TPL.FC_SetException(i_xExceptionActive	:= xUpdateStructsException, 
					iq_stException		:= stUpdateStructsException, 
					iq_stExceptionList	:= iq_stExceptionList, 
					iq_stLogDataList	:= iq_stLogDataList);
					
xInitSuccessful := xInitSuccessful AND NOT xUpdateStructsException;

etDiag := GD.ET_Diag.Ok;
(* End of system generated code, could be modified for your application *)
END_ACTION

END_PROGRAM

// LMC_PacDrive/Application/CrankModuleExample/Tools/FC_IsDriveVirtual
FUNCTION FC_IsDriveVirtual : BOOL
VAR_INPUT
	i_ifDrive	: SystemConfigurationItf.IF_Drive;
END_VAR

VAR_OUTPUT
	q_etDiag	: GD.ET_Diag := GD.ET_Diag.Ok;
	q_etDiagExt	: ET_DiagExt := ET_DiagExt.Ok;
	q_sMsg		: STRING[80];
END_VAR

VAR
	xSuccess						: BOOL;
	ifSercosDeviceIdentification	: SystemConfigurationItf.IF_SercosDeviceIdentification; 
END_VAR

IF i_ifDrive = 0 THEN
	q_etDiag	:= GD.ET_Diag.InputParameterInvalid;
	q_etDiagExt	:= ET_DiagExt.DriveInvalid;
	q_sMsg		:= 'FC_IsDriveVirtual: i_ifDrive not set';		
ELSE
	xSuccess := __QUERYINTERFACE(i_ifDrive, ifSercosDeviceIdentification);
	IF NOT xSuccess OR ifSercosDeviceIdentification = 0 THEN
		q_etDiag	:= GD.ET_Diag.InputParameterInvalid;
		q_etDiagExt	:= ET_DiagExt.DriveInvalid;
		q_sMsg		:= Standard.CONCAT(i_ifDrive.Name, ' - IF_SercosDeviceIdentification not implemented');						
	ELSE
		IF ifSercosDeviceIdentification.WorkingState = 0 THEN	// Drive is virtual
			FC_IsDriveVirtual := TRUE;
		ELSE
			FC_IsDriveVirtual := FALSE;
		END_IF
	END_IF
END_IF

END_FUNCTION

// LMC_PacDrive/Application/CrankModuleExample/Tools/FC_SetDeadTimeCompensation
FUNCTION FC_SetDeadTimeCompensation : BOOL
VAR_INPUT
	i_stSubModuleInterfaceMain		: AXM.ST_Main;
END_VAR
VAR
(* Init related variables *)	
	stLogicalAddressMaster			: SystemConfigurationItf.ST_LogicalAddress;
	lrShaftRefDelay					: LREAL;
	lrPositionDelay					: LREAL; 
	diResult						: DINT;	

END_VAR

IF i_stSubModuleInterfaceMain.i_ifMaster <> 0 AND i_stSubModuleInterfaceMain.i_ifDrive <> 0 THEN	
	stLogicalAddressMaster := i_stSubModuleInterfaceMain.i_ifMaster.stLogicalAddress;
	IF (stLogicalAddressMaster.udiType = SYSTEMINTERFACE.P_ENC_TYPE.udiType) OR			(* Physical encoder *)
		(stLogicalAddressMaster.udiType = SYSTEMINTERFACE.INC_IN_TYPE.udiType) OR		(* Incremental	encoder *)
		(stLogicalAddressMaster.udiType = SYSTEMINTERFACE.V_ENC_TYPE.udiType) THEN		(* Virtual master encoder *)
		
		stLogicalAddressMaster := i_stSubModuleInterfaceMain.i_ifDrive.stLogicalAddress;
		stLogicalAddressMaster.udiParameterId := 16#00A2;
		diResult := SYSTEMINTERFACE.FC_GetParameter(i_stLogAdr	:= stLogicalAddressMaster,
													i_dwBuffer	:= ADR(lrShaftRefDelay),
													i_diSize	:= SIZEOF(lrShaftRefDelay));
		IF diResult = 0 THEN
			i_stSubModuleInterfaceMain.iq_lencEncoder.Delay := -lrShaftRefDelay;
		END_IF
	ELSIF (stLogicalAddressMaster.udiType = SYSTEMINTERFACE.INC_IN3_TYPE.udiType) THEN  (* IncIn via TM5 TM5SE1IC20005 *)
		stLogicalAddressMaster := i_stSubModuleInterfaceMain.i_ifDrive.stLogicalAddress;
		stLogicalAddressMaster.udiParameterId := 16#00A2;
		diResult := SYSTEMINTERFACE.FC_GetParameter(i_stLogAdr	:= stLogicalAddressMaster,
													i_dwBuffer	:= ADR(lrShaftRefDelay),
													i_diSize	:= SIZEOF(lrShaftRefDelay));
		IF diResult = 0 THEN
			i_stSubModuleInterfaceMain.iq_lencEncoder.Delay := -lrShaftRefDelay;
			stLogicalAddressMaster := i_stSubModuleInterfaceMain.i_ifMaster.stLogicalAddress;
			stLogicalAddressMaster.udiParameterId := 16#008E; 					(* Parameter PositionDelay of TM5SE1IC20005 *)
			diResult := SYSTEMINTERFACE.FC_GetParameter(i_stLogAdr	:= stLogicalAddressMaster,
														i_dwBuffer	:= ADR(lrPositionDelay),
														i_diSize	:= SIZEOF(lrPositionDelay));		
			IF diResult = 0 THEN
				i_stSubModuleInterfaceMain.iq_lencEncoder.Delay := -(lrShaftRefDelay + (-lrPositionDelay)) ;
			END_IF
		END_IF
	END_IF
END_IF

IF diResult = 0 THEN
	FC_SetDeadTimeCompensation := TRUE;
END_IF

END_FUNCTION

// LMC_PacDrive/Application/CrankModuleExample/EquipmentModules/SR_BravoModule
PROGRAM SR_BravoModule

VAR CONSTANT
(* Standard related constants *)
	c_udiNumberOfGroups				: UDINT := 3;			(* Maximum number of groups *)
	c_udiNumberOfGroupMembers		: UDINT := 10;			(* Maximum number of members per group *)

	c_udiNumberOfCmdTables			: UDINT := 8;			(* Must be the exact number of used CMDTables! *)
	c_udiNumberOfCmdSteps			: UDINT := 16;			(* Make sure that the number of commands/ Steps  that each table
																   contains does not exceed the c_diNumberOfCMDSteps variable.*)

(* Definition group of modules *)
	c_udiBravoGroup1				: UDINT := 2001;		(* Name of module group  1 *)
	c_udiBravoGroup2				: UDINT := 2002;		(* Name of module group  2 *)

(* System generated code, could be modified for your application *)
	c_udiNumberOfSubModules			: UDINT := 2;			(* Number of axis modules *)
	c_udiSlave1						: UDINT := 1;
	c_udiSlave2						: UDINT := 2;
(* End of system generated code, could be modified for your application *)
END_VAR

VAR (* User specific variables *)
	stSlave1Interface				: AXM.ST_ModuleInterface;
	fbSlave1Module					: AXM.FB_AxisModule;
	
	stSlave2Interface				: AXM.ST_ModuleInterface;
	fbSlave2Module					: FB_AxisModuleExtItf;
	
	fbAxisModuleController			: AXM.FB_AxisModuleController;
END_VAR

VAR_INPUT
(* Master of BravoModule *)
	i_ifMaster						: SystemConfigurationItf.IF_Master;
END_VAR

VAR_IN_OUT
(* TPL.ST_StandardModuleInterface *)	
	iq_stStandardModuleItf			: TPL.ST_StandardModuleInterface;
	
(* TPL.ST_StandardMotionInterface *)		
	iq_stStandardMotionItf			: TPL.ST_StandardMotionInterface;
	
(* ExceptionHandling and Logging *)	
	iq_stExceptionList				: TPL.ST_ExceptionList;
	iq_stLogDataList				: TPL.ST_LogDataList;
END_VAR

VAR
	xInitSuccessful : BOOL := TRUE;
		
(* Standard related variables *)
	astSubModuleInterface			: ARRAY[1..c_udiNumberOfSubModules] OF TPL.ST_StandardModuleInterface;		(* Interface to modules *)
	aaudiSubModuleGroups			: ARRAY[1..c_udiNumberOfGroups,1..c_udiNumberOfGroupMembers] OF UDINT;
	adwSubModuleAddInterfaces		: ARRAY[1..c_udiNumberOfSubModules] OF DWORD;

(* Modules related variables *)
	fbModuleController				: TPL.FB_ModuleController;
	etDiagModuleController			: GD.ET_Diag;
	etDiagExtModuleController		: TPL.ET_DiagExt;
	sMsgModuleController			: STRING[80];
	xWaitForStartStep				: BOOL;
	
	astListOfCmdTables				: ARRAY [1..c_udiNumberOfCmdTables] OF TPL.ST_CmdTable;
	udiTableIndex					: UDINT;
	udiStepIndex					: UDINT;
	diStep							: DINT;

	astPrepareTable					: ARRAY [1..c_udiNumberOfCmdSteps] OF TPL.ST_Cmd;		(* Relating  Cmd table *)
	astAutoTable					: ARRAY [1..c_udiNumberOfCmdSteps] OF TPL.ST_Cmd;		(* Relating  Cmd table *)
	astManualTable					: ARRAY [1..c_udiNumberOfCmdSteps] OF TPL.ST_Cmd;		(* Relating  Cmd table *)
	astHoldTable					: ARRAY [1..c_udiNumberOfCmdSteps] OF TPL.ST_Cmd;		(* Relating  Cmd table *)
	astStartTable					: ARRAY [1..c_udiNumberOfCmdSteps] OF TPL.ST_Cmd;		(* Relating  Cmd table *)
	astStopTable					: ARRAY [1..c_udiNumberOfCmdSteps] OF TPL.ST_Cmd;		(* Relating  Cmd table *)
	astBrakeReleaseTable			: ARRAY [1..c_udiNumberOfCmdSteps] OF TPL.ST_Cmd;		(* Relating  Cmd table *)
	astAbortTable					: ARRAY [1..c_udiNumberOfCmdSteps] OF TPL.ST_Cmd;		(* Relating  Cmd table *)

(* ExceptionHandling related variables *)
	fbExceptionHandler				: TPL.FB_ExceptionHandler;

	aetReactionTranslationMode		: ARRAY[1..c_udiNumberOfSubModules] OF TPL.ET_ReactionTranslationMode;
	aastReactionTranslationTable	: ARRAY[1..c_udiNumberOfSubModules,1..TPL.Gc_udiMaxNumberOfReactions] OF TPL.ST_Reaction;
	astReactionTranslationJobs		: ARRAY[1..c_udiNumberOfSubModules] OF TPL.ST_ReactionTranslationJobs;
	
(* Exception declaration *)
	stUserException1				: TPL.ST_Exception;
	stUserException2				: TPL.ST_Exception;
	xModuleUserException1			: BOOL;
	xModuleUserException2			: BOOL;
	
	stUpdateStructsException		: TPL.ST_Exception;
	xUpdateStructsException			: BOOL;
	
	stInitReactionsException		: TPL.ST_Exception;
	xInitReactionsException			: BOOL;
	
	stInitSubModulesException		: TPL.ST_Exception;
	xInitSubModulesException		: BOOL;
	
	stIsDriveVirtualException		: TPL.ST_Exception;
	xIsDriveVirtualException		: BOOL;

(* Logging related variables *)
	fbLogger						: TPL.FB_Logger;

(* OnlineChange related variables *)
	fbDetectOnlineChange			: TPL.FB_DetectOnlineChange;
	xDetectOnlineChangeActive		: BOOL; 
	xDetectOnlineChangeReady		: BOOL; 
	etDetectOnlineChangeDiag		: GD.ET_Diag;
	etDetectOnlineChangeDiagExt		: TPL.ET_DiagExt; 
	sDetectOnlineChangeMsg			: STRING[80];
	
(* Init related variables *)	
	stLogicalAddressMaster			: SystemConfigurationItf.ST_LogicalAddress;
	lrShaftRefDelay					: LREAL;
	diResult						: DINT;	
	
	xDriveIsVirtual					: BOOL;	
	
(* POU-Feedback related variables *)	
	etDiag			: GD.ET_Diag;
	etDiagExt		: ET_DiagExt;
	etDiagExtTPL	: TPL.ET_DiagExt;
	etDiagExtAXM	: AXM.ET_DiagExt;
	sMsgBuffer		: STRING[80];
END_VAR

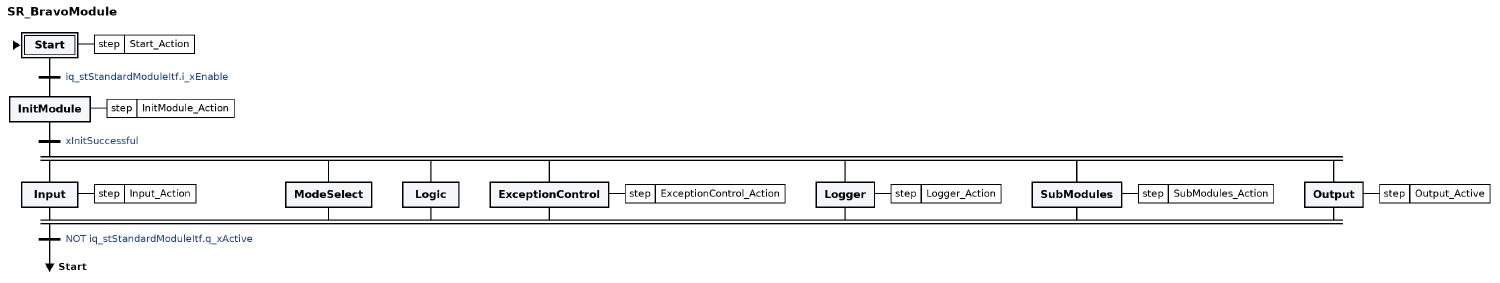
INITIAL_STEP Start:
    Start_Action(N);  // step action
END_STEP
TRANSITION FROM Start TO InitModule
    := iq_stStandardModuleItf.i_xEnable;
END_TRANSITION
STEP InitModule:
    InitModule_Action(N);  // step action
END_STEP
TRANSITION FROM InitModule TO (Input, ModeSelect, Logic, ExceptionControl, Logger, SubModules, Output)
    := xInitSuccessful;
END_TRANSITION
STEP Input:
    Input_Action(N);  // step action
END_STEP
STEP ModeSelect:
END_STEP
STEP Logic:
END_STEP
STEP ExceptionControl:
    ExceptionControl_Action(N);  // step action
END_STEP
STEP Logger:
    Logger_Action(N);  // step action
END_STEP
STEP SubModules:
    SubModules_Action(N);  // step action
END_STEP
STEP Output:
    Output_Active(N);  // step action
END_STEP
TRANSITION FROM (Input, ModeSelect, Logic, ExceptionControl, Logger, SubModules, Output) TO Start
    := NOT iq_stStandardModuleItf.q_xActive;
END_TRANSITION

ACTION ExceptionControl_Action:
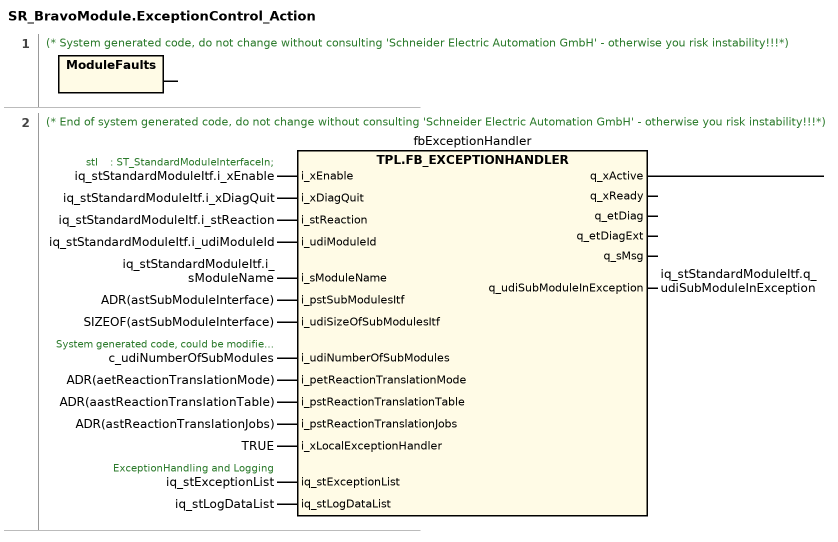
// NETWORK 1
// (* System generated code, do not change without consulting 'Schneider Electric Automation GmbH' - otherwise you risk instability!!!*)
ModuleFaults();

// NETWORK 2
// (* End of system generated code, do not change without consulting 'Schneider Electric Automation GmbH' - otherwise you risk instability!!!*)
//   fbExceptionHandler: ExceptionHandling related variables
//   iq_stStandardModuleItf.i_xEnable: stI : ST_StandardModuleInterfaceIn;
//   c_udiNumberOfSubModules: System generated code, could be modified for your application
//   iq_stExceptionList: ExceptionHandling and Logging
fbExceptionHandler(
    i_xEnable := iq_stStandardModuleItf.i_xEnable,
    i_xDiagQuit := iq_stStandardModuleItf.i_xDiagQuit,
    i_stReaction := iq_stStandardModuleItf.i_stReaction,
    i_udiModuleId := iq_stStandardModuleItf.i_udiModuleId,
    i_sModuleName := iq_stStandardModuleItf.i_sModuleName,
    i_pstSubModulesItf := ADR(astSubModuleInterface),
    i_udiSizeOfSubModulesItf := SIZEOF(astSubModuleInterface),
    i_udiNumberOfSubModules := c_udiNumberOfSubModules,
    i_petReactionTranslationMode := ADR(aetReactionTranslationMode),
    i_pstReactionTranslationTable := ADR(aastReactionTranslationTable),
    i_pstReactionTranslationJobs := ADR(astReactionTranslationJobs),
    i_xLocalExceptionHandler := TRUE,
    iq_stExceptionList := iq_stExceptionList,
    iq_stLogDataList := iq_stLogDataList,
    q_udiSubModuleInException => iq_stStandardModuleItf.q_udiSubModuleInException); // TPL.FB_EXCEPTIONHANDLER
END_ACTION

ACTION Init_CmdTables:
(* System generated code, could be modified for your application *)

(*********************************************************************************************************************)
(*** Prepare  ***)

TPL.FC_FirstStep(udiStepIndex, diStep);
astPrepareTable[udiStepIndex].sTitle					:= 'DriveEnable On AllSubModules';
astPrepareTable[udiStepIndex].udiModuleName				:= TPL.Gc_udiAllSubModules;
astPrepareTable[udiStepIndex].diStep					:= diStep;
astPrepareTable[udiStepIndex].diCMD						:= AXM.ET_Cmd.DriveEnableOn;
astPrepareTable[udiStepIndex].timTimeOut				:= T#0MS;
astPrepareTable[udiStepIndex].xEndCMD					:= FALSE;

TPL.FC_NextStep(udiStepIndex, diStep);
astPrepareTable[udiStepIndex].sTitle					:= 'Homing Mode AllSubModules';
astPrepareTable[udiStepIndex].udiModuleName				:= TPL.Gc_udiAllSubModules;
astPrepareTable[udiStepIndex].diStep					:= diStep;
astPrepareTable[udiStepIndex].diCMD						:= AXM.ET_Cmd.Homing;
astPrepareTable[udiStepIndex].timTimeOut				:= T#0MS;
astPrepareTable[udiStepIndex].xEndCMD					:= FALSE;

TPL.FC_NextStep(udiStepIndex, diStep);
astPrepareTable[udiStepIndex].sTitle					:= 'Homing Start AllSubModules';
astPrepareTable[udiStepIndex].udiModuleName				:= TPL.Gc_udiAllSubModules;
astPrepareTable[udiStepIndex].diStep					:= diStep;
astPrepareTable[udiStepIndex].diCMD						:= AXM.ET_Cmd.Start;
astPrepareTable[udiStepIndex].timTimeOut				:= T#0MS;
astPrepareTable[udiStepIndex].xEndCMD					:= FALSE;

TPL.FC_LastStep(udiStepIndex, diStep);
astPrepareTable[udiStepIndex].sTitle					:= 'End';
astPrepareTable[udiStepIndex].udiModuleName				:= 0;
astPrepareTable[udiStepIndex].diStep					:= diStep;
astPrepareTable[udiStepIndex].diCMD						:= 0;
astPrepareTable[udiStepIndex].timTimeOut				:= T#0MS;
astPrepareTable[udiStepIndex].xEndCMD					:= TRUE;

TPL.FC_FirstCmdTable(iq_udiTableIndex:= udiTableIndex);
astListofCMDTables[udiTableIndex].sTitle				:= 'Prepare';
astListofCMDTables[udiTableIndex].diCMD					:= ET_Cmd.Prepare;
astListofCMDTables[udiTableIndex].udiNumberOfCmdSteps	:= udiStepIndex;

(*********************************************************************************************************************)
(*** Auto  ***)

TPL.FC_FirstStep(udiStepIndex, diStep);
astAutoTable[udiStepIndex].sTitle						:= 'DriveEnable On AllSubModules';
astAutoTable[udiStepIndex].udiModuleName				:= TPL.Gc_udiAllSubModules;
astAutoTable[udiStepIndex].diStep						:= diStep;
astAutoTable[udiStepIndex].diCMD						:= AXM.ET_Cmd.DriveEnableOn;
astAutoTable[udiStepIndex].timTimeOut					:= T#0MS;
astAutoTable[udiStepIndex].xEndCMD						:= FALSE;

TPL.FC_NextStep(udiStepIndex, diStep);
astAutoTable[udiStepIndex].sTitle						:= 'Cam WS Mode AllSubModules';
astAutoTable[udiStepIndex].udiModuleName				:= TPL.Gc_udiAllSubModules;
astAutoTable[udiStepIndex].diStep						:= diStep;
astAutoTable[udiStepIndex].diCMD						:= AXM.ET_Cmd.CamWs;
astAutoTable[udiStepIndex].timTimeOut					:= T#0MS;
astAutoTable[udiStepIndex].xEndCMD						:= FALSE;

TPL.FC_NextStep(udiStepIndex, diStep);
astAutoTable[udiStepIndex].sTitle						:= 'Start AllSubModules';
astAutoTable[udiStepIndex].udiModuleName				:= TPL.Gc_udiAllSubModules;
astAutoTable[udiStepIndex].diStep						:= diStep;
astAutoTable[udiStepIndex].diCMD						:= AXM.ET_Cmd.Start;
astAutoTable[udiStepIndex].timTimeOut					:= T#0MS;
astAutoTable[udiStepIndex].xEndCMD						:= FALSE;

TPL.FC_NextStep(udiStepIndex, diStep);
astAutoTable[udiStepIndex].sTitle						:= 'WarmStart AllSubModules';
astAutoTable[udiStepIndex].udiModuleName				:= TPL.Gc_udiAllSubModules;
astAutoTable[udiStepIndex].diStep						:= diStep;
astAutoTable[udiStepIndex].diCMD						:= AXM.ET_Cmd.WsStart;
astAutoTable[udiStepIndex].timTimeOut					:= T#0MS;
astAutoTable[udiStepIndex].xEndCMD						:= FALSE;

TPL.FC_LastStep(udiStepIndex, diStep);
astAutoTable[udiStepIndex].sTitle						:= 'End';
astAutoTable[udiStepIndex].udiModuleName				:= 0;
astAutoTable[udiStepIndex].diStep						:= diStep;
astAutoTable[udiStepIndex].diCMD						:= 0;
astAutoTable[udiStepIndex].timTimeOut					:= T#0MS;
astAutoTable[udiStepIndex].xEndCMD						:= TRUE;

TPL.FC_NextCmdTable(iq_udiTableIndex:= udiTableIndex);
astListofCMDTables[udiTableIndex].sTitle				:= 'Auto';
astListofCMDTables[udiTableIndex].diCMD					:= ET_Cmd.Auto;
astListofCMDTables[udiTableIndex].udiNumberOfCmdSteps	:= udiStepIndex;

(*********************************************************************************************************************)
(*** Manual  ***)

TPL.FC_FirstStep(udiStepIndex, diStep);
astManualTable[udiStepIndex].sTitle						:= 'DriveEnable On AllSubModules';
astManualTable[udiStepIndex].udiModuleName				:= TPL.Gc_udiAllSubModules;
astManualTable[udiStepIndex].diStep						:= diStep;
astManualTable[udiStepIndex].diCMD						:= AXM.ET_Cmd.DriveEnableOn;
astManualTable[udiStepIndex].timTimeOut					:= T#0MS;
astManualTable[udiStepIndex].xEndCMD					:= FALSE;

TPL.FC_NextStep(udiStepIndex, diStep);
astManualTable[udiStepIndex].sTitle						:= 'Manual Mode AllSubModules';
astManualTable[udiStepIndex].udiModuleName				:= TPL.Gc_udiAllSubModules;
astManualTable[udiStepIndex].diStep						:= diStep;
astManualTable[udiStepIndex].diCMD						:= AXM.ET_Cmd.Manual;
astManualTable[udiStepIndex].timTimeOut					:= T#0MS;
astManualTable[udiStepIndex].xEndCMD					:= FALSE;

TPL.FC_LastStep(udiStepIndex, diStep);
astManualTable[udiStepIndex].sTitle						:= 'End';
astManualTable[udiStepIndex].udiModuleName				:= 0;
astManualTable[udiStepIndex].diStep						:= diStep;
astManualTable[udiStepIndex].diCMD						:= 0;
astManualTable[udiStepIndex].timTimeOut					:= T#0MS;
astManualTable[udiStepIndex].xEndCMD					:= TRUE;

TPL.FC_NextCmdTable(iq_udiTableIndex:= udiTableIndex);
astListofCMDTables[udiTableIndex].sTitle				:= 'Manual';
astListofCMDTables[udiTableIndex].diCMD					:= ET_Cmd.Manual;
astListofCMDTables[udiTableIndex].udiNumberOfCmdSteps	:= udiStepIndex;

(*********************************************************************************************************************)
(*** Stop ***)

TPL.FC_FirstStep(udiStepIndex, diStep);
astStopTable[udiStepIndex].sTitle						:= 'Stop AllSubModules';
astStopTable[udiStepIndex].udiModuleName				:= TPL.Gc_udiAllSubModules;
astStopTable[udiStepIndex].diStep						:= diStep;
astStopTable[udiStepIndex].diCMD						:= AXM.ET_Cmd.Stop;
astStopTable[udiStepIndex].timTimeOut					:= T#0MS;
astStopTable[udiStepIndex].xEndCMD						:= FALSE;

TPL.FC_LastStep(udiStepIndex, diStep);
astStopTable[udiStepIndex].sTitle						:= 'End';
astStopTable[udiStepIndex].udiModuleName				:= 0;
astStopTable[udiStepIndex].diStep						:= diStep;
astStopTable[udiStepIndex].diCMD						:= 0;
astStopTable[udiStepIndex].timTimeOut					:= T#0MS;
astStopTable[udiStepIndex].xEndCMD						:= TRUE;

TPL.FC_NextCmdTable(iq_udiTableIndex:= udiTableIndex);
astListofCMDTables[udiTableIndex].sTitle				:= 'Stop';
astListofCMDTables[udiTableIndex].diCMD					:= ET_Cmd.Stop;
astListofCMDTables[udiTableIndex].udiNumberOfCmdSteps	:= udiStepIndex;

(*********************************************************************************************************************)
(*** Start ***)

TPL.FC_FirstStep(udiStepIndex, diStep);
astStartTable[udiStepIndex].sTitle						:= 'Start AllSubModules';
astStartTable[udiStepIndex].udiModuleName				:= TPL.Gc_udiAllSubModules;
astStartTable[udiStepIndex].diStep						:= diStep;
astStartTable[udiStepIndex].diCMD						:= AXM.ET_Cmd.Start;
astStartTable[udiStepIndex].timTimeOut					:= T#0MS;
astStartTable[udiStepIndex].xEndCMD						:= FALSE;

TPL.FC_LastStep(udiStepIndex, diStep);
astStartTable[udiStepIndex].sTitle						:= 'End';
astStartTable[udiStepIndex].udiModuleName				:= 0;
astStartTable[udiStepIndex].diStep						:= diStep;
astStartTable[udiStepIndex].diCMD						:= 0;
astStartTable[udiStepIndex].timTimeOut					:= T#0MS;
astStartTable[udiStepIndex].xEndCMD						:= TRUE;

TPL.FC_NextCmdTable(iq_udiTableIndex:= udiTableIndex);
astListofCMDTables[udiTableIndex].sTitle				:= 'Start';
astListofCMDTables[udiTableIndex].diCMD					:= ET_Cmd.Start;
astListofCMDTables[udiTableIndex].udiNumberOfCmdSteps	:= udiStepIndex;

(*********************************************************************************************************************)
(*** Abort ***)

TPL.FC_FirstStep(udiStepIndex, diStep);
astAbortTable[udiStepIndex].sTitle						:= 'Stop AllSubModules';
astAbortTable[udiStepIndex].udiModuleName				:= TPL.Gc_udiAllSubModules;
astAbortTable[udiStepIndex].diStep						:= diStep;
astAbortTable[udiStepIndex].diCMD						:= AXM.ET_Cmd.Stop;
astAbortTable[udiStepIndex].timTimeOut					:= T#0MS;
astAbortTable[udiStepIndex].xEndCMD						:= FALSE;

TPL.FC_LastStep(udiStepIndex, diStep);
astAbortTable[udiStepIndex].sTitle						:= 	'End';
astAbortTable[udiStepIndex].udiModuleName				:= 	0;
astAbortTable[udiStepIndex].diStep						:= 	diStep;
astAbortTable[udiStepIndex].diCMD						:= 	0;
astAbortTable[udiStepIndex].timTimeOut					:=	T#0MS;
astAbortTable[udiStepIndex].xEndCMD						:= TRUE;

TPL.FC_NextCmdTable(iq_udiTableIndex:= udiTableIndex);
astListofCMDTables[udiTableIndex].sTitle				:= 'Abort';
astListofCMDTables[udiTableIndex].diCMD					:= ET_Cmd.Abort;
astListofCMDTables[udiTableIndex].udiNumberOfCmdSteps	:= udiStepIndex;

(*********************************************************************************************************************)
(*** Hold ***)

TPL.FC_FirstStep(udiStepIndex, diStep);
astHoldTable[udiStepIndex].sTitle						:= 'Hold AllSubModules';
astHoldTable[udiStepIndex].udiModuleName				:= TPL.Gc_udiAllSubModules;
astHoldTable[udiStepIndex].diStep						:= diStep;
astHoldTable[udiStepIndex].diCMD						:= AXM.ET_Cmd.Hold;
astHoldTable[udiStepIndex].timTimeOut					:= T#0MS;
astHoldTable[udiStepIndex].xEndCMD						:= FALSE;

TPL.FC_LastStep(udiStepIndex, diStep);
astHoldTable[udiStepIndex].sTitle						:= 'End';
astHoldTable[udiStepIndex].udiModuleName				:= 0;
astHoldTable[udiStepIndex].diStep						:= diStep;
astHoldTable[udiStepIndex].diCMD						:= 0;
astHoldTable[udiStepIndex].timTimeOut					:= T#0MS;
astHoldTable[udiStepIndex].xEndCMD						:= TRUE;

TPL.FC_NextCmdTable(iq_udiTableIndex:= udiTableIndex);
astListofCMDTables[udiTableIndex].sTitle				:= 'Hold';
astListofCMDTables[udiTableIndex].diCMD					:= ET_Cmd.Hold;
astListofCMDTables[udiTableIndex].udiNumberOfCmdSteps	:= udiStepIndex;

(*********************************************************************************************************************)
(*** Brake Release ***)

TPL.FC_FirstStep(udiStepIndex, diStep);
astBrakeReleaseTable[udiStepIndex].sTitle				:= 'AxisEnable Off AllSubModules';
astBrakeReleaseTable[udiStepIndex].udiModuleName		:= TPL.Gc_udiAllSubModules;
astBrakeReleaseTable[udiStepIndex].diStep				:= diStep;
astBrakeReleaseTable[udiStepIndex].diCMD				:= AXM.ET_Cmd.DriveEnableOff;
astBrakeReleaseTable[udiStepIndex].timTimeOut			:= T#0MS;
astBrakeReleaseTable[udiStepIndex].xEndCMD				:= FALSE;

TPL.FC_NextStep(udiStepIndex, diStep);
astBrakeReleaseTable[udiStepIndex].sTitle				:= 'BrakeRelease Mode AllSubModules';
astBrakeReleaseTable[udiStepIndex].udiModuleName		:= TPL.Gc_udiAllSubModules;
astBrakeReleaseTable[udiStepIndex].diStep				:= diStep;
astBrakeReleaseTable[udiStepIndex].diCMD				:= AXM.ET_Cmd.BrakeRelease;
astBrakeReleaseTable[udiStepIndex].timTimeOut			:= T#0MS;
astBrakeReleaseTable[udiStepIndex].xEndCMD				:= FALSE;

TPL.FC_NextStep(udiStepIndex, diStep);
astBrakeReleaseTable[udiStepIndex].sTitle				:= 'Start AllSubModules';
astBrakeReleaseTable[udiStepIndex].udiModuleName		:= TPL.Gc_udiAllSubModules;
astBrakeReleaseTable[udiStepIndex].diStep				:= diStep;
astBrakeReleaseTable[udiStepIndex].diCMD				:= AXM.ET_Cmd.Start;
astBrakeReleaseTable[udiStepIndex].timTimeOut			:= T#0MS;
astBrakeReleaseTable[udiStepIndex].xEndCMD				:= FALSE;

TPL.FC_LastStep(udiStepIndex, diStep);
astBrakeReleaseTable[udiStepIndex].sTitle				:= 'End';
astBrakeReleaseTable[udiStepIndex].udiModuleName		:= 0;
astBrakeReleaseTable[udiStepIndex].diStep				:= diStep;
astBrakeReleaseTable[udiStepIndex].diCMD				:= 0;
astBrakeReleaseTable[udiStepIndex].timTimeOut			:= T#0MS;
astBrakeReleaseTable[udiStepIndex].xEndCMD				:= TRUE;

TPL.FC_NextCmdTable(iq_udiTableIndex:= udiTableIndex);
astListofCMDTables[udiTableIndex].sTitle				:= 'Brake Release';
astListofCMDTables[udiTableIndex].diCMD					:= ET_Cmd.BrakeRelease;
astListofCMDTables[udiTableIndex].udiNumberOfCmdSteps	:= udiStepIndex;

(* End of system generated code, could be modified for your application *)
END_ACTION

ACTION Init_Exceptions:
(* System generated code, could be modified for your application *)
stUpdateStructsException.etDiag												:= GD.ET_Diag.UnexpectedProgramBehavior;
stUpdateStructsException.udiDiagExt											:= ET_DiagExt.UpdateStructsException;
stUpdateStructsException.sDiagExt											:= FC_EtDiagExtToString(i_etDiagExt := stUpdateStructsException.udiDiagExt);
stUpdateStructsException.sMsg												:= '';	(* Replaced on usage *)
stUpdateStructsException.udiModuleId										:= iq_stStandardModuleItf.i_udiModuleId;
stUpdateStructsException.sModuleName										:= iq_stStandardModuleItf.i_sModuleName;
stUpdateStructsException.stReaction.axReaction[TPL.ET_Reaction.AsyncStop]	:= TRUE;
stUpdateStructsException.etSource											:= TPL.ET_ExceptionSource.NodeModule;
stUpdateStructsException.timDelayTime										:= T#0MS;
stUpdateStructsException.wHmiAttributes										:= 0;
stUpdateStructsException.xAutoQuit											:= FALSE;

stInitReactionsException.etDiag												:= GD.ET_Diag.UnexpectedProgramBehavior;
stInitReactionsException.udiDiagExt											:= ET_DiagExt.InitReactionsException;
stInitReactionsException.sDiagExt											:= FC_EtDiagExtToString(i_etDiagExt := stInitReactionsException.udiDiagExt);
stInitReactionsException.sMsg												:= '';	(* Replaced on usage *)
stInitReactionsException.udiModuleId										:= iq_stStandardModuleItf.i_udiModuleId;
stInitReactionsException.sModuleName										:= iq_stStandardModuleItf.i_sModuleName;
stInitReactionsException.stReaction.axReaction[TPL.ET_Reaction.AsyncStop]	:= TRUE;
stInitReactionsException.etSource											:= TPL.ET_ExceptionSource.NodeModule;
stInitReactionsException.timDelayTime										:= T#0MS;
stInitReactionsException.wHmiAttributes										:= 0;
stInitReactionsException.xAutoQuit											:= FALSE;

stInitSubModulesException.etDiag											:= GD.ET_Diag.UnexpectedProgramBehavior;
stInitSubModulesException.udiDiagExt										:= ET_DiagExt.InitSubModulesException;
stInitSubModulesException.sDiagExt											:= FC_EtDiagExtToString(i_etDiagExt := stInitSubModulesException.udiDiagExt);
stInitSubModulesException.sMsg												:= '';	(* Replaced on usage *)
stInitSubModulesException.udiModuleId										:= iq_stStandardModuleItf.i_udiModuleId;
stInitSubModulesException.sModuleName										:= iq_stStandardModuleItf.i_sModuleName;
stInitSubModulesException.stReaction.axReaction[TPL.ET_Reaction.AsyncStop]	:= TRUE;
stInitSubModulesException.etSource											:= TPL.ET_ExceptionSource.NodeModule;
stInitSubModulesException.timDelayTime										:= T#0MS;
stInitSubModulesException.wHmiAttributes									:= 0;
stInitSubModulesException.xAutoQuit											:= FALSE;


(*------------------------------------------------------------------------------------------*)
(* Init User Exceptions *)

	// TPL.ET_Reaction.AsyncStop
	// TPL.ET_Reaction.SyncStopEL
	// TPL.ET_Reaction.SyncStopEH
	// TPL.ET_Reaction.StopEndOfCycle
	// TPL.ET_Reaction.MainsContactorOff
	
(*------------------------------------------------------------------------------------------*)
stUserException1.etDiag													:= GD.ET_Diag.ExecutionAborted;
stUserException1.udiDiagExt												:= ET_DiagExtUser.Exception1FromEquipmentModule;
stUserException1.sDiagExt												:= FC_EtDiagExtUserToString(i_etDiagExt := stUserException1.udiDiagExt);
stUserException1.sMsg													:= 'User Exception 1';
stUserException1.udiModuleId											:= iq_stStandardModuleItf.i_udiModuleId;
stUserException1.sModuleName											:= iq_stStandardModuleItf.i_sModuleName;
stUserException1.stReaction.axReaction[TPL.Gc_udiUserReactionOffset+2]	:= TRUE;
stUserException1.etSource												:= TPL.ET_ExceptionSource.User;
stUserException1.timDelayTime											:= T#0MS;
stUserException1.wHmiAttributes											:= 0;
stUserException1.xAutoQuit												:= FALSE;

stUserException2.etDiag													:= GD.ET_Diag.ExecutionAborted;
stUserException2.udiDiagExt												:= ET_DiagExtUser.Exception2FromEquipmentModule;
stUserException2.sDiagExt												:= FC_EtDiagExtUserToString(i_etDiagExt := stUserException2.udiDiagExt);
stUserException2.sMsg													:= 'User Exception 2';
stUserException2.udiModuleId											:= iq_stStandardModuleItf.i_udiModuleId;
stUserException2.sModuleName											:= iq_stStandardModuleItf.i_sModuleName;
stUserException2.stReaction.axReaction[TPL.Gc_udiUserReactionOffset+2]	:= TRUE;
stUserException2.etSource												:= TPL.ET_ExceptionSource.User;
stUserException2.timDelayTime											:= T#0MS;
stUserException2.wHmiAttributes											:= 0;
stUserException2.xAutoQuit												:= FALSE;

(* End of system generated code, could be modified for your application *)
END_ACTION

ACTION Init_Reactions:
(* System generated code, only to be changed by experienced programmers *)
IF c_udiNumberOfSubModules < 1 THEN
	RETURN;
END_IF

(* Change of default reactions only on demand *)
(* Compare SR MainMachine Action Init_Reactions *)

xInitReactionsException := FALSE;

(*****************************************************************************************************************************************************)
(* Init ReactionTranslationMode *)

TPL.FC_InitReactionTranslationMode(	i_udiNumberOfSubModules			:= c_udiNumberOfSubModules,
									i_petReactionTranslationMode	:= ADR(aetReactionTranslationMode),
									q_etDiag						=> etDiag,
									q_etDiagExt						=> etDiagExtTPL);
							
IF etDiag <> GD.ET_Diag.Ok AND NOT xInitReactionsException THEN
	xInitReactionsException := TRUE;
	
	stInitReactionsException.sMsg := PDL.FC_MultiConcat(i_sString1 := 'InitReactionTranslationMode - ', 
														i_sString2 := GD.FC_EtDiagToString(i_etDiag := etDiag), 
														i_sString3 := ' - ', 
														i_sString4 := TPL.FC_EtDiagExtToString(i_etDiagExt := etDiagExtTPL));
END_IF	

(*****************************************************************************************************************************************************)
(* Init ReactionTranslationTable *)	

TPL.FC_InitReactionTranslationTable(i_udiNumberOfSubModules			:= c_udiNumberOfSubModules,
									i_pstReactionTranslationTable	:= ADR(aastReactionTranslationTable),
									q_etDiag						=> etDiag,
									q_etDiagExt						=> etDiagExtTPL);
									
IF etDiag <> GD.ET_Diag.Ok AND NOT xInitReactionsException THEN
	xInitReactionsException := TRUE;
	
	stInitReactionsException.sMsg := PDL.FC_MultiConcat(i_sString1 := 'InitReactionTranslationTable - ', 
														i_sString2 := GD.FC_EtDiagToString(i_etDiag := etDiag), 
														i_sString3 := ' - ', 
														i_sString4 := TPL.FC_EtDiagExtToString(i_etDiagExt := etDiagExtTPL));
END_IF		

(*****************************************************************************************************************************************************)
(* Init ReactionTranslationJobs *)	
								
TPL.FC_InitReactionTranslationJobs( i_udiNumberOfSubModules			:= c_udiNumberOfSubModules,
									i_pstReactionTranslationJobs	:= ADR(astReactionTranslationJobs),
									q_etDiag						=> etDiag,
									q_etDiagExt						=> etDiagExtTPL);
						
IF etDiag <> GD.ET_Diag.Ok AND NOT xInitReactionsException THEN
	xInitReactionsException := TRUE;
	
	stInitReactionsException.sMsg := PDL.FC_MultiConcat(i_sString1 := 'InitReactionTranslationJobs - ', 
														i_sString2 := GD.FC_EtDiagToString(i_etDiag := etDiag), 
														i_sString3 := ' - ', 
														i_sString4 := TPL.FC_EtDiagExtToString(i_etDiagExt := etDiagExtTPL));
END_IF		

(*****************************************************************************************************************************************************)
(* Set exception if any exception occurred *)

TPL.FC_SetException(i_xExceptionActive	:= xInitReactionsException, 
					iq_stException		:= stInitReactionsException, 
					iq_stExceptionList	:= iq_stExceptionList, 
					iq_stLogDataList	:= iq_stLogDataList);
					
xInitSuccessful := xInitSuccessful AND NOT xInitReactionsException;

etDiag := GD.ET_Diag.Ok;
(* End of system generated code, only to be changed by experienced programmers *)
END_ACTION

ACTION Init_Slave1:
(* System generated code, could be modified for your application *)

(* Standard interface *)
astSubModuleInterface[c_udiSlave1].i_sModuleName		:= CONCAT(STR1 := iq_stStandardModuleItf.i_sModuleName, STR2 := ': Slave1');

astSubModuleInterface[c_udiSlave1].i_xLogEnable			:= 	TRUE;
astSubModuleInterface[c_udiSlave1].i_wLogDataFilter		:= 	UDINT_TO_WORD(TPL.ET_LogDataFilter.ModuleDefault);

(* AxisModule specific interface *)
stSlave1Interface.stMain.i_ifMaster			:= i_ifMaster; 		(* Master *)
stSlave1Interface.stMain.i_ifDrive			:= DRV_Slave1;
stSlave1Interface.stMain.iq_lencEncoder		:= LE_Slave1;


xDriveIsVirtual := FC_IsDriveVirtual(	i_ifDrive	:= stSlave1Interface.stMain.i_ifDrive,
										q_etDiag	=> etDiag,
										q_etDiagExt	=> etDiagExt, //etDiagExtTPL,
										q_sMsg		=> sMsgBuffer);

IF etDiag <> GD.ET_Diag.Ok AND NOT xIsDriveVirtualException THEN										
	stIsDriveVirtualException.sMsg := sMsgBuffer;
	xIsDriveVirtualException := TRUE;
END_IF

TPL.FC_SetException(i_xExceptionActive	:= xIsDriveVirtualException, 
					iq_stException		:= stIsDriveVirtualException, 
					iq_stExceptionList	:= iq_stExceptionList, 
					iq_stLogDataList	:= iq_stLogDataList);
					
xInitSuccessful := xInitSuccessful AND NOT xIsDriveVirtualException;
etDiag := GD.ET_Diag.Ok;
	

(*Set DeadTime compensation parameters depending on used type of Master*)
FC_SetDeadTimeCompensation(i_stSubModuleInterfaceMain := stSlave1Interface.stMain);
  (*Please note, FC_DeadTimeCompensation does not recognize the master type, transferred via C2C or encoder network! 
	stXXXXInterface.stMain.iq_lencEncoder.Delay must be adjusted in order to reach shaft synchronism, it depends on:
	- Transmission delay via the choosen network, depending on topology and timing 
	- Type of the master e.g. physical encoder or an axis
	- SERCOS cycle times in master and slave controllers
	
	C2C sample (similar for encoder network):
	//Access C2C_EncIn.DataDelay only if C2C_Master.SyncGroupState=5 or C2C_Slave.SyncGroupState = 5 and C2C_EncIn.DataValid = TRUE!

		//Master is a physical encoder (PMEnc/Inc):
			stXXXXInterface.stMain.iq_lencEncoder.Delay := C2C_EncIn.DataDelay - DRV_SlaveAxis.ShaftRefDelay;

		//Master is an axis (real/ virtual):
			stXXXXInterface.stMain.iq_lencEncoder.Delay := C2C_EncIn.DataDelay + one SERCOS cycle of C2C controller with connected master axis;*)


stSlave1Interface.stMain.i_lrMotionActiveVelLimit						:= 15.0;	(* Limit for max. velocity of astAxisModuleInterface to switch output AxisMove in Units/s *)
stSlave1Interface.stMain.i_etMotionActiveVelType						:= AXM.ET_MotionActiveVelType.Velocity;

stSlave1Interface.stMain.i_timMasterStop								:= T#1S;
stSlave1Interface.stMain.i_xHwLimitPos									:= FALSE;
stSlave1Interface.stMain.i_xHwLimitNeg									:= FALSE;

stSlave1Interface.stMain.stReducedVelocity.i_xEnableReducedVelocity		:= FALSE;
stSlave1Interface.stMain.stReducedVelocity.i_xOnlyLimitCheck			:= FALSE;
stSlave1Interface.stMain.stReducedVelocity.i_lrMaxReducedVelocity		:= 50.0;

stSlave1Interface.stMain.i_xStart										:= FALSE;

(***************************************************************************************************************************************************************************************************)

(*** Homing ***)

IF xDriveIsVirtual THEN
	stSlave1Interface.stHome.i_etMode := PDL.ET_HomeMode.SetPosAxisAndLogEncoderPosition;			(* Homing Mode  in case of virtual axis *)
ELSE
	stSlave1Interface.stHome.i_etMode := PDL.ET_HomeMode.PosDirectionPosEdgeTp;						(* Homing Mode in case of real axis *)
END_IF
	

stSlave1Interface.stHome.i_xEnableInitAbsReadPos := FALSE;		(* TRUE : Restores the AxisPosition depending on the stHome.etMode
																		  If stHome.i_etMode is equal to PDL.ET_HomeMode.RestorePosFromAxisEncoder or 
																		  to PDL.ET_HomeMode.WriteAxisEncoder, the encoder of the axis is read,
																		  or else the position will be restored from the retain area *)
																		  
stSlave1Interface.stHome.stSetpos.iq_pstRestorePosRetain := ADR(Grp_stRestorePositionAxis2);

stSlave1Interface.stHome.i_xResetHomeOk := FALSE;

(* Possible modes for homing mode Sensor:
	PDL.ET_HomeMode.PosDirectionPosEdgeSensor
	PDL.ET_HomeMode.NegDirectionPosEdgeSensor
	PDL.ET_HomeMode.NegDirectionNegEdgeSensor
	PDL.ET_HomeMode.PosDirectionNegEdgeSensor
*)
stSlave1Interface.stHome.stSensor.i_lrHomePosition			:= 0.0;			(* Position at the end of homing in units *)
stSlave1Interface.stHome.stSensor.i_lrVel					:= 10.0;		(* Homing ceiling velocity in units/s *)
stSlave1Interface.stHome.stSensor.i_lrAcc					:= 1000.0;		(* Homing acceleration in units/s^2 *)
stSlave1Interface.stHome.stSensor.i_lrDec					:= 1000.0;		(* Homing deceleration in units/s^2 *)
stSlave1Interface.stHome.stSensor.i_lrJerk					:= 10000.0;		(* Homing jerk in units/s^3 *)
stSlave1Interface.stHome.stSensor.i_lrOffset				:= 0.0;			(* Offset from home signal in units *)
stSlave1Interface.stHome.stSensor.i_lrMaxTravel				:= 720.0;		(* Max. travel for referencing by normal input *)
stSlave1Interface.stHome.stSensor.i_xRotativeSystem			:= FALSE;		(* Rotative system true or false for referencing by normal input *)
stSlave1Interface.stHome.stSensor.i_xSensor					:= FALSE;		(* Input for home signal. Can be a signal from a controller input. Has to be written cyclic. *)

(* Possible Modes for homing mode LimitSwitch:
	PDL.ET_HomeMode.PosDirectionPosEdgeHWLimitPos		normally open contact / Closing contact
	PDL.ET_HomeMode.NegDirectionPosEdgeHWLimitNeg		normally open contact / Closing contact
	PDL.ET_HomeMode.NegDirectionNegEdgeHWLimitNeg		normally closed contact / Opening contact  
	PDL.ET_HomeMode.PosDirectionNegEdgeHWLimitPos		normally closed contact / Opening contact 
*)
stSlave1Interface.stHome.stLimitSwitch.i_lrHomePosition		:= 0.0;			(* Position at the end of homing in units *)
stSlave1Interface.stHome.stLimitSwitch.i_lrVel				:= 10.0;		(* Homing ceiling velocity in units/s *)
stSlave1Interface.stHome.stLimitSwitch.i_lrLowVel			:= 5.0;			(* Homing low ceiling velocity in units/s *)
stSlave1Interface.stHome.stLimitSwitch.i_lrAcc				:= 1000.0;		(* Homing acceleration in units/s^2 *)
stSlave1Interface.stHome.stLimitSwitch.i_lrDec				:= 1000.0;		(* Homing deceleration in units/s^2 *)
stSlave1Interface.stHome.stLimitSwitch.i_lrJerk				:= 10000.0;		(* Homing jerk in units/s^3 *)
stSlave1Interface.stHome.stLimitSwitch.i_lrOffset			:= 0.0;			(* Offset from home signal in units *)
stSlave1Interface.stHome.stLimitSwitch.i_lrMaxTravel		:= 9999.0;		(* Max. travel for referencing normal input as a hardware limit *)

(* Possible modes for homing mode MoveOnPos:
	PDL.ET_HomeMode.MoveOnPosAbs 
*)
stSlave1Interface.stHome.stMoveOnPos.i_lrTarget				:= 0.0;			(* Position at the end of homing in units *)
stSlave1Interface.stHome.stMoveOnPos.i_lrVel				:= 10.0;		(* Homing ceiling velocity in units/s *)
stSlave1Interface.stHome.stMoveOnPos.i_lrAcc				:= 1000.0;		(* Homing acceleration in units/s^2 *)
stSlave1Interface.stHome.stMoveOnPos.i_lrDec				:= 1000.0;		(* Homing deceleration in units/s^2 *)
stSlave1Interface.stHome.stMoveOnPos.i_lrJerk				:= 10000.0;		(* Homing jerk in units/s^3 *)
stSlave1Interface.stHome.stMoveOnPos.i_lrPeriod				:= 0.0;			(* Period of the axis *)
stSlave1Interface.stHome.stMoveOnPos.i_xRotativeSystem		:= FALSE;		(* Rotative system true or false *)

(* Possible modes for homing mode SetPos:
	PDL.ET_HomeMode.SetPosAxisPosition 
	PDL.ET_HomeMode.SetPosLogEncoderPosition 
	PDL.ET_HomeMode.SetPosAxisAndLogEncoderPosition
	PDL.ET_HomeMode.RestorePosFromAxisEncoder 
	PDL.ET_HomeMode.RestorePosFromRetain 
*)
stSlave1Interface.stHome.stSetpos.i_lrHomePosition			:= 0.0;			(* Position at the end of homing in units *)
stSlave1Interface.stHome.stSetpos.i_lrEncoderPosition		:= 0.0;			(* Encoder position in units after homing *)
stSlave1Interface.stHome.stSetpos.i_lrAbsEncOffset			:= 100.0;		(* Distance to the jump of axis encoder in units  *)
stSlave1Interface.stHome.stSetpos.i_lrRestoreWindow			:= 180;			(* How far can the drive be away from is correct position *)
stSlave1Interface.stHome.stSetpos.i_lrUserPeriod			:= 360;			(* Period of the axis *)

(* Possible modes for homing mode Torque:
	PDL.ET_HomeMode.PosDirectionMaxTorque 
	PDL.ET_HomeMode.NegDirectionMaxTorque 
*)
stSlave1Interface.stHome.stTorque.i_lrHomePosition			:= 0.0;			(* Position at the end of homing in units *)
stSlave1Interface.stHome.stTorque.i_lrVel					:= 10.0;		(* Homing ceiling velocity in units/s *)
stSlave1Interface.stHome.stTorque.i_lrAcc					:= 1000.0;		(* Homing acceleration in units/s^2 *)
stSlave1Interface.stHome.stTorque.i_lrDec					:= 1000.0;		(* Homing deceleration in units/s^2 *)
stSlave1Interface.stHome.stTorque.i_lrJerk					:= 10000.0;		(* Homing jerk in units/s^3 *)
stSlave1Interface.stHome.stTorque.i_lrOffset				:= 0.0;			(* Offset from home signal in units *)
stSlave1Interface.stHome.stTorque.i_lrMaxTravel				:= 9999.0;		(* Max. travel for referencing by torque *)
stSlave1Interface.stHome.stTorque.i_lrMaxTorque				:= 0.0;			(* Torque for stop in Nm / referencing by torque *)
stSlave1Interface.stHome.stTorque.i_diTorqueTime			:= 5;			(* Time in msec to hold torque *)

(* Possible modes for homing mode TouchProbe:
	PDL.ET_HomeMode.PosDirectionPosEdgeTp 
	PDL.ET_HomeMode.NegDirectionPosEdgeTp 
	PDL.ET_HomeMode.NegDirectionNegEdgeTp 
	PDL.ET_HomeMode.PosDirectionNegEdgeTp 
*)
stSlave1Interface.stHome.stTouchProbe.i_lrHomePosition		:= 0.0;			(* Position at the end of homing in units *)
stSlave1Interface.stHome.stTouchProbe.i_lrVel				:= 100.0;		(* Homing ceiling velocity in units/s *)
stSlave1Interface.stHome.stTouchProbe.i_lrAcc				:= 1000.0;		(* Homing acceleration in units/s^2 *)
stSlave1Interface.stHome.stTouchProbe.i_lrDec				:= 1000.0;		(* Homing deceleration in units/s^2 *)
stSlave1Interface.stHome.stTouchProbe.i_lrJerk				:= 10000.0;		(* Homing jerk in units/s^3 *)
stSlave1Interface.stHome.stTouchProbe.i_lrOffset			:= 30.0;		(* Offset from home signal in units *)
stSlave1Interface.stHome.stTouchProbe.i_lrMaxTravel			:= 720.0;		(* Max. travel for referencing by TP *)
stSlave1Interface.stHome.stTouchProbe.i_xRotativeSystem		:= TRUE;		(* Rotative system true or false for referencing by TP *)
stSlave1Interface.stHome.stTouchProbe.i_ifTouchProbe		:= TP_1;		(* Input for TP *)

(* Possible modes for homing mode WritePos:
	PDL.ET_HomeMode.WriteAxisEncoder 
*)
stSlave1Interface.stHome.stWritePos.i_lrHomePosition		:= 0.0;			(* Position at the end of homing in units *)
stSlave1Interface.stHome.stWritePos.i_lrUserPeriod			:= 0.0;			(* Calculates Drive.Position into period ( units ) *)
stSlave1Interface.stHome.stWritePos.i_lrAbsEncOffset		:= 100.0;		(* Distance to the jump of axis encoder in units *)

(***************************************************************************************************************************************************************************************************)
(*** Manual ***)

stSlave1Interface.stManual.i_lrVel								:= 50.0;			(* Velocity in units/s *)
stSlave1Interface.stManual.i_lrAcc								:= 100.0;			(* Acceleration in units/s^2 *)
stSlave1Interface.stManual.i_lrDec								:= 100.0;			(* Deceleration in units/s^2 *)
stSlave1Interface.stManual.i_lrJerk								:= 1000.0;			(* Jerk in units/s^3 *)
stSlave1Interface.stManual.i_lrMaxDistance						:= 120.0;			(* Max pathlengths for one step in units *)
stSlave1Interface.stManual.i_xEndless							:= FALSE;			(* TRUE: jogging endless; Position between the periode; FALSE: jogging in steps. Position can be out of periode *)
stSlave1Interface.stManual.i_lrPeriod							:= 360.0;			(* Period of the axis *)

(***************************************************************************************************************************************************************************************************)
(*** Cam ***)

stSlave1Interface.stMultiCam.i_etCSModeSlave					:= PDL.ET_MultiCamCsModeSlave.SetSlavePositionToFirstCamPosition;		(* ColdStartMode Slave *)
stSlave1Interface.stMultiCam.i_etCSModeMaster					:= PDL.ET_MultiCamCsModeMaster.SetMasterPositionToFirstCamPosition;		(* ColdStartMode Master *)
stSlave1Interface.stMultiCam.i_etWSMode							:= PDL.ET_MultiCamWsMode.StoredCamMoveAlwaysNoPositionCheck;			(* WarmStartMode *)
stSlave1Interface.stMultiCam.i_lrWSWindow						:= 5.0;											(* WarmStartWindow in Axis units *)
stSlave1Interface.stMultiCam.i_lrWSVel							:= 100.0;										(* Velocity for WarmStart and CSModeSlave = PDL.ET_MultiCamCsModeSlave.MoveSlaveToFirstCamPosition in Units/s *)
stSlave1Interface.stMultiCam.i_lrWSAcc							:= 1000.0;										(* Acceleration and deceleration for Warmstart and CSModeSlave = PDL.ET_MultiCamCsModeSlave.MoveSlaveToFirstCamPosition in Units/s^2 *)
stSlave1Interface.stMultiCam.i_lrWSJerk							:= 10000.0;										(* Jerk for Warmstart and CSModeSlave = PDL.ET_MultiCamCsModeSlave.MoveSlaveToFirstCamPosition in units/s^3 *)
stSlave1Interface.stMultiCam.i_diTXend							:= 2*SYSTEMINTERFACE.FC_LzsTaskGetInterval();	(* Time of XLowEnd and XHighEnd befor Xend or Xstart in msec*)
stSlave1Interface.stMultiCam.i_lrInstantXLimMax					:= 0.0;											(* Switch off position at 'InstantNewCam' *)

stSlave1Interface.stMultiCam.i_xEnableTabHandler				:= TRUE;										(* TRUE: TabHandler is enabled *)
stSlave1Interface.stMultiCam.i_udiTableSelectNr					:= AXM.ET_ParId.User;							(* Number of table which is used in the next cycle *)

stSlave1Interface.stMultiCam.i_xSetEncoderParameters			:= FALSE;										(* TRUE: The parameters MasterId, FeedConstand, GearIn and GearOut will be copyed into LEnc object *)
stSlave1Interface.stMultiCam.i_xSetEncoderPosition				:= FALSE;										(* TRUE: Manipulation of LEnc object on startup OpMode MultiCam *)
stSlave1Interface.stMultiCam.i_lrSetEncoderOffset				:= 0.0;											(* Master encoder offset *)
stSlave1Interface.stMultiCam.i_xCheckEncoderPeriod				:= TRUE;										(* TRUE: Check of encoder period = 0. If encoder period <> 0 -> Exception *)

stSlave1Interface.stMultiCam.iq_astMotionPar[AXM.ET_ParId.User].diNumberOfCamPoints		:= 4;	(* DataStruct for the next cycle *)
stSlave1Interface.stMultiCam.iq_astMotionPar[AXM.ET_ParId.User].lrYPeriod				:= 0.0;

stSlave1Interface.stMultiCam.iq_astMotionPar[AXM.ET_ParId.User].astCamPoint[0].lrX		:= 0.0;
stSlave1Interface.stMultiCam.iq_astMotionPar[AXM.ET_ParId.User].astCamPoint[0].lrY		:= 0.0;
stSlave1Interface.stMultiCam.iq_astMotionPar[AXM.ET_ParId.User].astCamPoint[0].lrM		:= 0.0;
stSlave1Interface.stMultiCam.iq_astMotionPar[AXM.ET_ParId.User].astCamPoint[0].etCamType	:= PDL.ET_CamType.Poly5Com;
stSlave1Interface.stMultiCam.iq_astMotionPar[AXM.ET_ParId.User].astCamPoint[1].lrX		:= 60.0;
stSlave1Interface.stMultiCam.iq_astMotionPar[AXM.ET_ParId.User].astCamPoint[1].lrY		:= 30.0;
stSlave1Interface.stMultiCam.iq_astMotionPar[AXM.ET_ParId.User].astCamPoint[1].lrM		:= 1.0;
stSlave1Interface.stMultiCam.iq_astMotionPar[AXM.ET_ParId.User].astCamPoint[1].etCamType	:= PDL.ET_CamType.Straight;
stSlave1Interface.stMultiCam.iq_astMotionPar[AXM.ET_ParId.User].astCamPoint[2].lrX		:= 240.0;
stSlave1Interface.stMultiCam.iq_astMotionPar[AXM.ET_ParId.User].astCamPoint[2].lrY		:= 210.0;
stSlave1Interface.stMultiCam.iq_astMotionPar[AXM.ET_ParId.User].astCamPoint[2].lrM		:= 1.0;
stSlave1Interface.stMultiCam.iq_astMotionPar[AXM.ET_ParId.User].astCamPoint[2].etCamType	:= PDL.ET_CamType.Poly5Com;
stSlave1Interface.stMultiCam.iq_astMotionPar[AXM.ET_ParId.User].astCamPoint[3].lrX		:= 360.0;
stSlave1Interface.stMultiCam.iq_astMotionPar[AXM.ET_ParId.User].astCamPoint[3].lrY		:= 0.0;
stSlave1Interface.stMultiCam.iq_astMotionPar[AXM.ET_ParId.User].astCamPoint[3].lrM		:= 0.0;
stSlave1Interface.stMultiCam.iq_astMotionPar[AXM.ET_ParId.User].astCamPoint[3].etCamType	:= PDL.ET_CamType.Poly5Com;

stSlave1Interface.stMultiCam.iq_astMotionPar[AXM.ET_ParId.Idle].diUserTableId	:= UDINT_TO_DINT(AXM.ET_ParId.Idle);
stSlave1Interface.stMultiCam.iq_astMotionPar[AXM.ET_ParId.Start].diUserTableId	:= UDINT_TO_DINT(AXM.ET_ParId.Start);
stSlave1Interface.stMultiCam.iq_astMotionPar[AXM.ET_ParId.Cont].diUserTableId	:= UDINT_TO_DINT(AXM.ET_ParId.Cont);
stSlave1Interface.stMultiCam.iq_astMotionPar[AXM.ET_ParId.Stop].diUserTableId	:= UDINT_TO_DINT(AXM.ET_ParId.Stop);
stSlave1Interface.stMultiCam.iq_astMotionPar[AXM.ET_ParId.User].diUserTableId	:= UDINT_TO_DINT(AXM.ET_ParId.User);

(***************************************************************************************************************************************************************************************************)
(*** Endless ***)

stSlave1Interface.stEndless.i_lrVel								:= 100.0;			(* Velocity in Units/s *)
stSlave1Interface.stEndless.i_lrAcc								:= 1000.0;			(* Acceleration in Units/s^2 *)
stSlave1Interface.stEndless.i_lrDec								:= 1000.0;			(* Deceleration in Units/s^2 *)
stSlave1Interface.stEndless.i_lrJerk							:= 10000.0;			(* Jerk in units/s^3 *)
stSlave1Interface.stEndless.i_lrPeriod							:= 360.0;			(* Period one cycle in units *)
stSlave1Interface.stEndless.i_lrStopPosition					:= 0.5;				(* Stop position in units *)


(***************************************************************************************************************************************************************************************************)
(*** Pos ***)

stSlave1Interface.stPos.i_etPosMode								:= SYSTEMINTERFACE.ET_PosMode.Relative;			(* SYSTEMINTERFACE.ET_PosMode.Endless, SYSTEMINTERFACE.ET_PosMode.Relative, SYSTEMINTERFACE.ET_PosMode.Absolute *)
stSlave1Interface.stPos.i_lrTarget								:= -360.0;										(* Target position or distance in Units *)
stSlave1Interface.stPos.i_lrVel									:= 100.0;										(* Ceiling velocity in Units/s *)
stSlave1Interface.stPos.i_lrAcc									:= 3600.0;										(* Acceleration in Units/s^2 *)
stSlave1Interface.stPos.i_lrDec									:= 3600.0;										(* Deceleration in Units/s^2 *)
stSlave1Interface.stPos.i_lrJerk								:= 36000.0;										(* Jerk in units/s^3 *)

(* End of system generated code, could be modified for your application *)
END_ACTION

ACTION Init_Slave2:
(* System generated code, could be modified for your application *)

(* Standard interface *)
astSubModuleInterface[c_udiSlave2].i_sModuleName	:= 	CONCAT(STR1 := iq_stStandardModuleItf.i_sModuleName, STR2 := ': Slave2');

astSubModuleInterface[c_udiSlave2].i_xLogEnable		:= 	TRUE;
astSubModuleInterface[c_udiSlave2].i_wLogDataFilter	:= 	UDINT_TO_WORD(TPL.ET_LogDataFilter.ModuleDefault);

(* AxisModule specific interface *)
stSlave2Interface.stMain.i_ifMaster		:= i_ifMaster; 		(* Master *)
stSlave2Interface.stMain.i_ifDrive		:= DRV_Slave2;
stSlave2Interface.stMain.iq_lencEncoder	:= LE_Slave2;


xDriveIsVirtual := FC_IsDriveVirtual(	i_ifDrive	:= stSlave2Interface.stMain.i_ifDrive,
										q_etDiag	=> etDiag,
										q_etDiagExt	=> etDiagExt,//etDiagExtTPL,
										q_sMsg		=> sMsgBuffer);

IF etDiag <> GD.ET_Diag.Ok AND NOT xIsDriveVirtualException THEN										
	stIsDriveVirtualException.sMsg := sMsgBuffer;
	xIsDriveVirtualException := TRUE;
END_IF

TPL.FC_SetException(i_xExceptionActive	:= xIsDriveVirtualException, 
					iq_stException		:= stIsDriveVirtualException, 
					iq_stExceptionList	:= iq_stExceptionList, 
					iq_stLogDataList	:= iq_stLogDataList);
					
xInitSuccessful := xInitSuccessful AND NOT xIsDriveVirtualException;
etDiag := GD.ET_Diag.Ok;
	

(*Set DeadTime compensation parameters depending on used type of Master*)
FC_SetDeadTimeCompensation(i_stSubModuleInterfaceMain := stSlave2Interface.stMain);
  (*Please note, FC_DeadTimeCompensation does not recognize the master type, transferred via C2C or encoder network! 
	stXXXXInterface.stMain.iq_lencEncoder.Delay must be adjusted in order to reach shaft synchronism, it depends on:
	- Transmission delay via the choosen network, depending on topology and timing 
	- Type of the master e.g. physical encoder or an axis
	- SERCOS cycle times in master and slave controllers
	
	C2C sample (similar for encoder network):
	//Access C2C_EncIn.DataDelay only if C2C_Master.SyncGroupState=5 or C2C_Slave.SyncGroupState = 5 and C2C_EncIn.DataValid = TRUE!

		//Master is a physical encoder (PMEnc/Inc):
			stXXXXInterface.stMain.iq_lencEncoder.Delay := C2C_EncIn.DataDelay - DRV_SlaveAxis.ShaftRefDelay;

		//Master is an axis (real/ virtual):
			stXXXXInterface.stMain.iq_lencEncoder.Delay := C2C_EncIn.DataDelay + one SERCOS cycle of C2C controller with connected master axis;*)


stSlave2Interface.stMain.i_lrMotionActiveVelLimit						:= 15.0;	(* Limit for max. velocity of astAxisModuleInterface to switch output AxisMove in Units/s *)
stSlave2Interface.stMain.i_etMotionActiveVelType						:= AXM.ET_MotionActiveVelType.Velocity;

stSlave2Interface.stMain.i_timMasterStop								:= T#1S;
stSlave2Interface.stMain.i_xHwLimitPos									:= FALSE;
stSlave2Interface.stMain.i_xHwLimitNeg									:= FALSE;

stSlave2Interface.stMain.stReducedVelocity.i_xEnableReducedVelocity		:= FALSE;
stSlave2Interface.stMain.stReducedVelocity.i_xOnlyLimitCheck			:= FALSE;
stSlave2Interface.stMain.stReducedVelocity.i_lrMaxReducedVelocity		:= 50.0;

stSlave2Interface.stMain.i_xStart										:= FALSE;

(***************************************************************************************************************************************************************************************************)

(*** Homing ***)

IF xDriveIsVirtual THEN
	stSlave2Interface.stHome.i_etMode := PDL.ET_HomeMode.SetPosAxisAndLogEncoderPosition;			(* Homing Mode  in case of virtual axis *)
ELSE
	stSlave2Interface.stHome.i_etMode := PDL.ET_HomeMode.PosDirectionPosEdgeTp;						(* Homing Mode in case of real axis *)
END_IF


stSlave2Interface.stHome.i_xEnableInitAbsReadPos := FALSE;		(* TRUE : Restores the AxisPosition depending on the stHome.etMode
																		  If stHome.i_etMode is equal to PDL.ET_HomeMode.RestorePosFromAxisEncoder or 
																		  to PDL.ET_HomeMode.WriteAxisEncoder, the encoder of the axis is read,
																		  or else the position will be restored from the retain area *)
																								 
stSlave2Interface.stHome.stSetpos.iq_pstRestorePosRetain := ADR(Grp_stRestorePositionAxis3);

stSlave2Interface.stHome.i_xResetHomeOk := FALSE;

(* Possible modes for homing mode Sensor:
	PDL.ET_HomeMode.PosDirectionPosEdgeSensor
	PDL.ET_HomeMode.NegDirectionPosEdgeSensor
	PDL.ET_HomeMode.NegDirectionNegEdgeSensor
	PDL.ET_HomeMode.PosDirectionNegEdgeSensor
*)
stSlave2Interface.stHome.stSensor.i_lrHomePosition			:= 0.0;			(* Position at the end of homing in units *)
stSlave2Interface.stHome.stSensor.i_lrVel					:= 10.0;		(* Homing ceiling velocity in units/s *)
stSlave2Interface.stHome.stSensor.i_lrAcc					:= 1000.0;		(* Homing acceleration in units/s^2 *)
stSlave2Interface.stHome.stSensor.i_lrDec					:= 1000.0;		(* Homing deceleration in units/s^2 *)
stSlave2Interface.stHome.stSensor.i_lrJerk					:= 10000.0;		(* Homing jerk in units/s^3 *)
stSlave2Interface.stHome.stSensor.i_lrOffset				:= 0.0;			(* Offset from home signal in units *)
stSlave2Interface.stHome.stSensor.i_lrMaxTravel				:= 720.0;		(* Max. travel for referencing by normal input *)
stSlave2Interface.stHome.stSensor.i_xRotativeSystem			:= FALSE;		(* Rotative system true or false for referencing by normal input *)
stSlave2Interface.stHome.stSensor.i_xSensor					:= FALSE;		(* Input for home signal. Can be a signal from a controller input. Has to be written cyclic. *)

(* Possible Modes for homing mode LimitSwitch:
	PDL.ET_HomeMode.PosDirectionPosEdgeHWLimitPos		normally open contact / Closing contact
	PDL.ET_HomeMode.NegDirectionPosEdgeHWLimitNeg		normally open contact / Closing contact
	PDL.ET_HomeMode.NegDirectionNegEdgeHWLimitNeg		normally closed contact / Opening contact  
	PDL.ET_HomeMode.PosDirectionNegEdgeHWLimitPos		normally closed contact / Opening contact 
*)
stSlave2Interface.stHome.stLimitSwitch.i_lrHomePosition		:= 0.0;			(* Position at the end of homing in units *)
stSlave2Interface.stHome.stLimitSwitch.i_lrVel				:= 10.0;		(* Homing ceiling velocity in units/s *)
stSlave2Interface.stHome.stLimitSwitch.i_lrLowVel			:= 5.0;			(* Homing low ceiling velocity in units/s *)
stSlave2Interface.stHome.stLimitSwitch.i_lrAcc				:= 1000.0;		(* Homing acceleration in units/s^2 *)
stSlave2Interface.stHome.stLimitSwitch.i_lrDec				:= 1000.0;		(* Homing deceleration in units/s^2 *)
stSlave2Interface.stHome.stLimitSwitch.i_lrJerk				:= 10000.0;		(* Homing jerk in units/s^3 *)	
stSlave2Interface.stHome.stLimitSwitch.i_lrOffset			:= 0.0;			(* Offset from home signal in units *)
stSlave2Interface.stHome.stLimitSwitch.i_lrMaxTravel		:= 9999.0;		(* Max. travel for referencing normal input as a hardware limit *)

(* Possible modes for homing mode MoveOnPos:
	PDL.ET_HomeMode.MoveOnPosAbs 
*)
stSlave2Interface.stHome.stMoveonPos.i_lrTarget				:= 0.0;			(* Position at the end of homing in units *)
stSlave2Interface.stHome.stMoveonPos.i_lrVel				:= 10.0;		(* Homing ceiling velocity in units/s *)
stSlave2Interface.stHome.stMoveonPos.i_lrAcc				:= 1000.0;		(* Homing acceleration in units/s^2 *)
stSlave2Interface.stHome.stMoveonPos.i_lrDec				:= 1000.0;		(* Homing deceleration in units/s^2 *)
stSlave2Interface.stHome.stMoveonPos.i_lrJerk				:= 10000.0;		(* Homing jerk in units/s^3 *)
stSlave2Interface.stHome.stMoveonPos.i_lrPeriod				:= 0.0;			(* Period of the axis *)
stSlave2Interface.stHome.stMoveonPos.i_xRotativeSystem		:= FALSE;		(* Rotative system true or false *)

(* Possible modes for homing mode SetPos:
	PDL.ET_HomeMode.SetPosAxisPosition 
	PDL.ET_HomeMode.SetPosLogEncoderPosition 
	PDL.ET_HomeMode.SetPosAxisAndLogEncoderPosition
	PDL.ET_HomeMode.RestorePosFromAxisEncoder 
	PDL.ET_HomeMode.RestorePosFromRetain 
*)
stSlave2Interface.stHome.stSetpos.i_lrHomePosition			:= 0.0;			(* Position at the end of homing in units *)
stSlave2Interface.stHome.stSetpos.i_lrEncoderPosition		:= 0.0;			(* Encoder position in units after homing *)
stSlave2Interface.stHome.stSetpos.i_lrAbsEncOffset			:= 100.0;		(* Distance to the jump of axis encoder in units  *)
stSlave2Interface.stHome.stSetpos.i_lrRestoreWindow			:= 180;			(* How far can the drive be away from is correct position *)
stSlave2Interface.stHome.stSetpos.i_lrUserPeriod			:= 360;			(* Period of the axis *)

(* Possible modes for homing mode Torque:
	PDL.ET_HomeMode.PosDirectionMaxTorque 
	PDL.ET_HomeMode.NegDirectionMaxTorque 
*)
stSlave2Interface.stHome.stTorque.i_lrHomePosition			:= 0.0;			(* Position at the end of homing in units *)
stSlave2Interface.stHome.stTorque.i_lrVel					:= 10.0;		(* Homing ceiling velocity in units/s *)
stSlave2Interface.stHome.stTorque.i_lrAcc					:= 1000.0;		(* Homing acceleration in units/s^2 *)
stSlave2Interface.stHome.stTorque.i_lrDec					:= 1000.0;		(* Homing deceleration in units/s^2 *)
stSlave2Interface.stHome.stTorque.i_lrJerk					:= 10000.0;		(* Homing jerk in units/s^3 *)
stSlave2Interface.stHome.stTorque.i_lrOffset				:= 0.0;			(* Offset from home signal in units *)
stSlave2Interface.stHome.stTorque.i_lrMaxTravel				:= 9999.0;		(* Max. travel for referencing by torque *)
stSlave2Interface.stHome.stTorque.i_lrMaxTorque				:= 0.0;			(* Torque for stop in Nm / referencing by torque *)
stSlave2Interface.stHome.stTorque.i_diTorqueTime			:= 5;			(* Time in msec to hold torque *)

(* Possible modes for homing mode TouchProbe:
	PDL.ET_HomeMode.PosDirectionPosEdgeTp 
	PDL.ET_HomeMode.NegDirectionPosEdgeTp 
	PDL.ET_HomeMode.NegDirectionNegEdgeTp 
	PDL.ET_HomeMode.PosDirectionNegEdgeTp 
*)
stSlave2Interface.stHome.stTouchProbe.i_lrHomePosition		:= 0.0;			(* Position at the end of homing in units *)
stSlave2Interface.stHome.stTouchProbe.i_lrVel				:= 100.0;		(* Homing ceiling velocity in units/s *)
stSlave2Interface.stHome.stTouchProbe.i_lrAcc				:= 1000.0;		(* Homing acceleration in units/s^2 *)
stSlave2Interface.stHome.stTouchProbe.i_lrDec				:= 1000.0;		(* Homing deceleration in units/s^2 *)
stSlave2Interface.stHome.stTouchProbe.i_lrJerk				:= 10000.0;		(* Homing jerk in units/s^3 *)
stSlave2Interface.stHome.stTouchProbe.i_lrOffset			:= 30.0;		(* Offset from home signal in units *)
stSlave2Interface.stHome.stTouchProbe.i_lrMaxTravel			:= 720.0;		(* Max. travel for referencing by TP *)
stSlave2Interface.stHome.stTouchProbe.i_xRotativeSystem		:= TRUE;		(* Rotative system true or false for referencing by TP *)
stSlave2Interface.stHome.stTouchProbe.i_ifTouchProbe		:= TP_2;		(* Input for TP *)

(* Possible modes for homing mode WritePos:
	PDL.ET_HomeMode.WriteAxisEncoder 
*)
stSlave2Interface.stHome.stWritePos.i_lrHomePosition		:= 0.0;			(* Position at the end of homing in units *)
stSlave2Interface.stHome.stWritePos.i_lrUserPeriod			:= 0.0;			(* Calculates Drive.position into period ( units ) *)
stSlave2Interface.stHome.stWritePos.i_lrAbsEncOffset		:= 100.0;		(* Distance to the jump of axis encoder in units *)

(***************************************************************************************************************************************************************************************************)
(*** Manual ***)

stSlave2Interface.stManual.i_lrVel								:= 50.0;			(* Velocity in units/s *)
stSlave2Interface.stManual.i_lrAcc								:= 100.0;			(* Acceleration in units/s^2 *)
stSlave2Interface.stManual.i_lrDec								:= 100.0;			(* Deceleration in units/s^2 *)
stSlave2Interface.stManual.i_lrJerk								:= 1000.0;			(* Jerk in units/s^3 *)
stSlave2Interface.stManual.i_lrMaxDistance						:= 120.0;			(* Max pathlengths for one step in units *)
stSlave2Interface.stManual.i_xEndless							:= FALSE;			(* TRUE: jogging endless; Position between the periode; FALSE: jogging in steps. Position can be out of periode *)
stSlave2Interface.stManual.i_lrPeriod							:= 360.0;			(* Period of the axis *)

(***************************************************************************************************************************************************************************************************)
(*** Cam ***)

stSlave2Interface.stMultiCam.i_etCSModeSlave					:= PDL.ET_MultiCamCsModeSlave.SetSlavePositionToFirstCamPosition;		(* ColdStartMode Slave *)
stSlave2Interface.stMultiCam.i_etCSModeMaster					:= PDL.ET_MultiCamCsModeMaster.SetMasterPositionToFirstCamPosition;		(* ColdStartMode Master *)
stSlave2Interface.stMultiCam.i_etWSMode							:= PDL.ET_MultiCamWsMode.StoredCamMoveAlwaysNoPositionCheck;			(* WarmStartMode *)
stSlave2Interface.stMultiCam.i_lrWSWindow						:= 5.0;											(* WarmStartWindow in Axis units *)
stSlave2Interface.stMultiCam.i_lrWSVel							:= 100.0;										(* Velocity for WarmStart and CSModeSlave = PDL.ET_MultiCamCsModeSlave.MoveSlaveToFirstCamPosition in Units/s *)
stSlave2Interface.stMultiCam.i_lrWSAcc							:= 1000.0;										(* Acceleration and deceleration for Warmstart and CSModeSlave = PDL.ET_MultiCamCsModeSlave.MoveSlaveToFirstCamPosition in Units/s^2 *)
stSlave2Interface.stMultiCam.i_lrWSJerk							:= 10000.0;										(* Jerk for Warmstart and CSModeSlave = PDL.ET_MultiCamCsModeSlave.MoveSlaveToFirstCamPosition in units/s^3 *)
stSlave2Interface.stMultiCam.i_diTXend							:= 2*SYSTEMINTERFACE.FC_LzsTaskGetInterval();	(* Time of XLowEnd and XHighEnd befor Xend or Xstart in msec*)
stSlave2Interface.stMultiCam.i_lrInstantXLimMax					:= 0.0;											(* Switch off position at 'InstantNewCam' *)

stSlave2Interface.stMultiCam.i_xEnableTabHandler				:= TRUE;										(* TRUE: TabHandler is enabled *)
stSlave2Interface.stMultiCam.i_udiTableSelectNr					:= AXM.ET_ParId.User;							(* Number of table which is used in the next cycle *)								

stSlave2Interface.stMultiCam.i_xSetEncoderParameters			:= FALSE;										(* TRUE: The parameters MasterId, FeedConstand, GearIn and GearOut will be copyed into LEnc object *)
stSlave2Interface.stMultiCam.i_xSetEncoderPosition				:= FALSE;										(* TRUE: Manipulation of LEnc object on startup OpMode MultiCam *)
stSlave2Interface.stMultiCam.i_lrSetEncoderOffset				:= 0.0;											(* Master encoder offset *)
stSlave2Interface.stMultiCam.i_xCheckEncoderPeriod				:= TRUE;										(* TRUE: Check of encoder period = 0. If encoder period <> 0 -> Exception *)

stSlave2Interface.stMultiCam.iq_astMotionPar[AXM.ET_ParId.User].diNumberOfCamPoints		:= 4;	(* DataStruct for the next cycle *)
stSlave2Interface.stMultiCam.iq_astMotionPar[AXM.ET_ParId.User].lrYPeriod				:= 0.0;

stSlave2Interface.stMultiCam.iq_astMotionPar[AXM.ET_ParId.User].astCamPoint[0].lrX		:= 0.0;
stSlave2Interface.stMultiCam.iq_astMotionPar[AXM.ET_ParId.User].astCamPoint[0].lrY		:= 0.0;
stSlave2Interface.stMultiCam.iq_astMotionPar[AXM.ET_ParId.User].astCamPoint[0].lrM		:= 0.0;
stSlave2Interface.stMultiCam.iq_astMotionPar[AXM.ET_ParId.User].astCamPoint[0].etCamType	:= PDL.ET_CamType.Poly5Com;
stSlave2Interface.stMultiCam.iq_astMotionPar[AXM.ET_ParId.User].astCamPoint[1].lrX		:= 60.0;
stSlave2Interface.stMultiCam.iq_astMotionPar[AXM.ET_ParId.User].astCamPoint[1].lrY		:= 30.0;
stSlave2Interface.stMultiCam.iq_astMotionPar[AXM.ET_ParId.User].astCamPoint[1].lrM		:= 1.0;
stSlave2Interface.stMultiCam.iq_astMotionPar[AXM.ET_ParId.User].astCamPoint[1].etCamType	:= PDL.ET_CamType.Straight;
stSlave2Interface.stMultiCam.iq_astMotionPar[AXM.ET_ParId.User].astCamPoint[2].lrX		:= 240.0;
stSlave2Interface.stMultiCam.iq_astMotionPar[AXM.ET_ParId.User].astCamPoint[2].lrY		:= 210.0;
stSlave2Interface.stMultiCam.iq_astMotionPar[AXM.ET_ParId.User].astCamPoint[2].lrM		:= 1.0;
stSlave2Interface.stMultiCam.iq_astMotionPar[AXM.ET_ParId.User].astCamPoint[2].etCamType	:= PDL.ET_CamType.Poly5Com;
stSlave2Interface.stMultiCam.iq_astMotionPar[AXM.ET_ParId.User].astCamPoint[3].lrX		:= 360.0;
stSlave2Interface.stMultiCam.iq_astMotionPar[AXM.ET_ParId.User].astCamPoint[3].lrY		:= 0.0;
stSlave2Interface.stMultiCam.iq_astMotionPar[AXM.ET_ParId.User].astCamPoint[3].lrM		:= 0.0;
stSlave2Interface.stMultiCam.iq_astMotionPar[AXM.ET_ParId.User].astCamPoint[3].etCamType	:= PDL.ET_CamType.Poly5Com;

stSlave2Interface.stMultiCam.iq_astMotionPar[AXM.ET_ParId.Idle].diUserTableId	:= UDINT_TO_DINT(AXM.ET_ParId.Idle);
stSlave2Interface.stMultiCam.iq_astMotionPar[AXM.ET_ParId.Start].diUserTableId	:= UDINT_TO_DINT(AXM.ET_ParId.Start);
stSlave2Interface.stMultiCam.iq_astMotionPar[AXM.ET_ParId.Cont].diUserTableId	:= UDINT_TO_DINT(AXM.ET_ParId.Cont);
stSlave2Interface.stMultiCam.iq_astMotionPar[AXM.ET_ParId.Stop].diUserTableId	:= UDINT_TO_DINT(AXM.ET_ParId.Stop);
stSlave2Interface.stMultiCam.iq_astMotionPar[AXM.ET_ParId.User].diUserTableId	:= UDINT_TO_DINT(AXM.ET_ParId.User);


(***************************************************************************************************************************************************************************************************)
(*** Endless ***)

stSlave2Interface.stEndless.i_lrVel								:= 100.0;			(* Velocity in Units/s *)
stSlave2Interface.stEndless.i_lrAcc								:= 1000.0;			(* Acceleration in Units/s^2 *)
stSlave2Interface.stEndless.i_lrDec								:= 1000.0;			(* Deceleration in Units/s^2 *)
stSlave2Interface.stEndless.i_lrJerk							:= 10000.0;			(* Jerk in units/s^3 *)
stSlave2Interface.stEndless.i_lrPeriod							:= 360.0;			(* Period one cycle in units *)
stSlave2Interface.stEndless.i_lrStopPosition					:= 0.5;				(* Stop position in units *)


(***************************************************************************************************************************************************************************************************)
(*** Pos ***)

stSlave2Interface.stPos.i_etPosMode								:= SYSTEMINTERFACE.ET_PosMode.Relative;		(* SYSTEMINTERFACE.ET_PosMode.Endless, SYSTEMINTERFACE.ET_PosMode.Relative, SYSTEMINTERFACE.ET_PosMode.Absolute *)
stSlave2Interface.stPos.i_lrTarget								:= 360.0;									(* Target position or distance in Units *)
stSlave2Interface.stPos.i_lrVel									:= 3600.0;									(* Ceiling velocity in Units/s *)
stSlave2Interface.stPos.i_lrAcc									:= 36000.0;									(* Acceleration in Units/s^2 *)
stSlave2Interface.stPos.i_lrDec									:= 36000.0;									(* Deceleration in Units/s^2 *)
stSlave2Interface.stPos.i_lrJerk								:= 360000.0;								(* Jerk in units/s^3 *)

(* End of system generated code, could be modified for your application *)
END_ACTION

ACTION Init_SubModules:
(* System generated code, could be modified for your application *)

(*** Module Group declaration ***)

aaudiSubModuleGroups[c_udiBravoGroup1-TPL.Gc_udiGroupOffset,TPL.ET_Group.Member1] := 0;				(* There is no first element of the group c_diBravoGroup1 *)
aaudiSubModuleGroups[c_udiBravoGroup1-TPL.Gc_udiGroupOffset,TPL.ET_Group.Member2] := 0;				(* There is no second element of the group c_diBravoGroup1 *)

aaudiSubModuleGroups[c_udiBravoGroup2-TPL.Gc_udiGroupOffset,TPL.ET_Group.Member1] := c_udiSlave1;		(* The Slave1 is the first element of the group c_diBravoGroup2 *)
aaudiSubModuleGroups[c_udiBravoGroup2-TPL.Gc_udiGroupOffset,TPL.ET_Group.Member2] := c_udiSlave2;		(* The Slave2 is the second element of the group c_diBravoGroup2 *)

(* End of system generated code, could be modified for your application *)


(* System generated code, do not change without consulting 'Schneider Electric Automation GmbH' - otherwise you risk instability!!!*)
xInitSubModulesException := FALSE;

(*****************************************************************************************************************************************************)
(* Set IDs of SubModules *)	

TPL.FC_SetSubModuleIds(	i_udiMainModuleID			:= iq_stStandardModuleItf.i_udiModuleId,
						i_pstSubModulesItf			:= ADR(astSubModuleInterface),
						i_udiNumberOfSubModules		:= c_udiNumberOfSubModules,
						q_etDiag					=> etDiag,
						q_etDiagExt					=> etDiagExtTPL);

IF etDiag <> GD.ET_Diag.Ok AND NOT xInitSubModulesException THEN
	xInitSubModulesException := TRUE;
	
	stInitSubModulesException.sMsg := PDL.FC_MultiConcat(	i_sString1 := 'SetSubModuleIds - ', 
															i_sString2 := GD.FC_EtDiagToString(i_etDiag := etDiag), 
															i_sString3 := ' - ', 
															i_sString4 := TPL.FC_EtDiagExtToString(i_etDiagExt := etDiagExtTPL));
END_IF	

(*****************************************************************************************************************************************************)
(* Set exception if any exception occurred *)

TPL.FC_SetException(i_xExceptionActive	:= xInitSubModulesException, 
					iq_stException		:= stInitSubModulesException, 
					iq_stExceptionList	:= iq_stExceptionList, 
					iq_stLogDataList	:= iq_stLogDataList);

xInitSuccessful := xInitSuccessful AND NOT xInitSubModulesException;
					
etDiag := GD.ET_Diag.Ok;
(* End of system generated code, do not change without consulting 'Schneider Electric Automation GmbH' - otherwise you risk instability!!!*)
END_ACTION

ACTION InitModule_Action:
(* This step is used for initialisations after being enabled *)

(* System generated code, could be modified for your application *)
xInitSuccessful := TRUE;

Init_Exceptions();
(* End of system generated code, could be modified for your application *)

(* System generated code, do not change without consulting 'Schneider Electric Automation GmbH' - otherwise you risk instability!!!*)
iq_stStandardModuleItf.q_xActive			:= TRUE;
iq_stStandardModuleItf.q_xReady			:= FALSE;
iq_stStandardModuleItf.q_etDiag			:= GD.ET_Diag.Ok;
iq_stStandardModuleItf.q_udiDiagExt		:= ET_DiagExt.Initializing;
iq_stStandardModuleItf.q_sDiagExt			:= FC_EtDiagExtToString(i_etDiagExt := ET_DiagExt.Initializing);
iq_stStandardModuleItf.q_sMsg				:= '';

Init_SubModules();
Init_CmdTables();
Init_Reactions();
UpdateStructs();
(* End of system generated code, do not change without consulting 'Schneider Electric Automation GmbH' - otherwise you risk instability!!!*)

(* System generated code, could be modified for your application *)
Init_Slave1();
Init_Slave2();
(* End of system generated code, could be modified for your application *)

(* Application specific code *)
(* ToDo: Add your application specific code here *)
;
(* End of application specific code *)
END_ACTION

ACTION Input_Action:
(* System generated code, do not change without consulting 'Schneider Electric Automation GmbH' - otherwise you risk instability!!!*)
UpdateStructs();
(* End of system generated code, do not change without consulting 'Schneider Electric Automation GmbH' - otherwise you risk instability!!!*)
END_ACTION

ACTION Logger_Action:
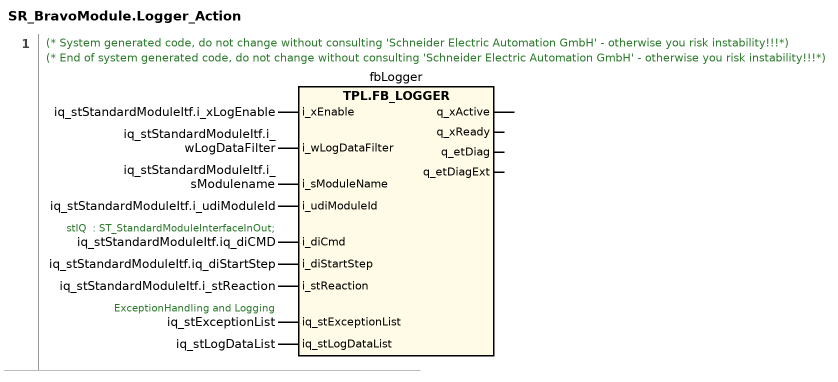
// NETWORK 1
// 					(* System generated code, do not change without consulting 'Schneider Electric Automation GmbH' - otherwise you risk instability!!!*)
// (* End of system generated code, do not change without consulting 'Schneider Electric Automation GmbH' - otherwise you risk instability!!!*)
//
//   fbLogger: Logging related variables
//   iq_stStandardModuleItf.iq_diCMD: stIQ : ST_StandardModuleInterfaceInOut;
//   iq_stExceptionList: ExceptionHandling and Logging
fbLogger(
    i_xEnable := iq_stStandardModuleItf.i_xLogEnable,
    i_wLogDataFilter := iq_stStandardModuleItf.i_wLogDataFilter,
    i_sModuleName := iq_stStandardModuleItf.i_sModulename,
    i_udiModuleId := iq_stStandardModuleItf.i_udiModuleId,
    i_diCmd := iq_stStandardModuleItf.iq_diCMD,
    i_diStartStep := iq_stStandardModuleItf.iq_diStartStep,
    i_stReaction := iq_stStandardModuleItf.i_stReaction,
    iq_stExceptionList := iq_stExceptionList,
    iq_stLogDataList := iq_stLogDataList); // TPL.FB_LOGGER
END_ACTION

ACTION ModuleFaults:
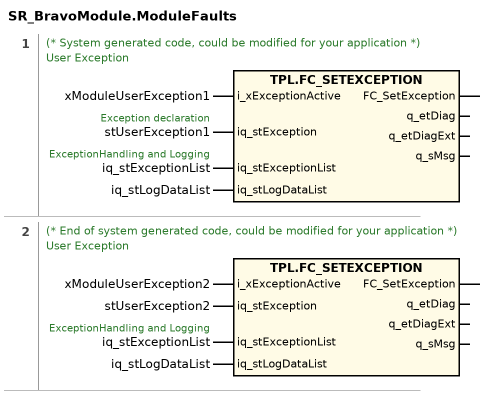
// NETWORK 1
// (* System generated code, could be modified for your application *)
// User Exception
//   stUserException1: Exception declaration
//   iq_stExceptionList: ExceptionHandling and Logging
TPL.FC_SETEXCEPTION(i_xExceptionActive := xModuleUserException1, iq_stException := stUserException1, iq_stExceptionList := iq_stExceptionList, iq_stLogDataList := iq_stLogDataList);

// NETWORK 2
// (* End of system generated code, could be modified for your application *)
// User Exception
//   iq_stExceptionList: ExceptionHandling and Logging
TPL.FC_SETEXCEPTION(i_xExceptionActive := xModuleUserException2, iq_stException := stUserException2, iq_stExceptionList := iq_stExceptionList, iq_stLogDataList := iq_stLogDataList);
END_ACTION

ACTION Output_Active:
(* System generated code, only to be changed by experienced programmers *)
IF iq_stStandardModuleItf.q_udiSubModuleInException <> 0 THEN
	iq_stStandardModuleItf.q_etDiag		:= GD.ET_Diag.Ok;
	iq_stStandardModuleItf.q_udiDiagExt	:= ET_DiagExt.SubModuleInException;
	iq_stStandardModuleItf.q_sDiagExt		:= FC_EtDiagExtToString(i_etDiagExt := ET_DiagExt.SubModuleInException);
	iq_stStandardModuleItf.q_sMsg			:= '';
ELSE
	IF etDiagModuleController = GD.ET_Diag.Ok THEN
		iq_stStandardModuleItf.q_etDiag	:= etDiagModuleController;
		iq_stStandardModuleItf.q_sMsg		:= sMsgModuleController;
		
		CASE etDiagExtModuleController OF
			TPL.ET_DiagExt.DeactivatingSubModules : 
				iq_stStandardModuleItf.q_udiDiagExt	:= ET_DiagExt.DeactivatingSubModules;
				iq_stStandardModuleItf.q_sDiagExt		:= FC_EtDiagExtToString(i_etDiagExt := ET_DiagExt.DeactivatingSubModules);
			TPL.ET_DiagExt.Disabled : 
				iq_stStandardModuleItf.q_udiDiagExt	:= ET_DiagExt.Disabled;
				iq_stStandardModuleItf.q_sDiagExt		:= FC_EtDiagExtToString(i_etDiagExt := ET_DiagExt.Disabled);
			TPL.ET_DiagExt.ExecuteStep : 
				iq_stStandardModuleItf.q_udiDiagExt	:= ET_DiagExt.ExecuteStep;
				iq_stStandardModuleItf.q_sDiagExt		:= FC_EtDiagExtToString(i_etDiagExt := ET_DiagExt.ExecuteStep);
			TPL.ET_DiagExt.Initializing : 
				iq_stStandardModuleItf.q_udiDiagExt	:= ET_DiagExt.Initializing;
				iq_stStandardModuleItf.q_sDiagExt		:= FC_EtDiagExtToString(i_etDiagExt := ET_DiagExt.Initializing);
			TPL.ET_DiagExt.WaitAtNegativeStep : 
				iq_stStandardModuleItf.q_udiDiagExt	:= ET_DiagExt.WaitAtNegativeStep;
				iq_stStandardModuleItf.q_sDiagExt		:= FC_EtDiagExtToString(i_etDiagExt := ET_DiagExt.WaitAtNegativeStep);
			TPL.ET_DiagExt.WaitCmdsDone : 
				iq_stStandardModuleItf.q_udiDiagExt	:= ET_DiagExt.WaitCmdsDone;
				iq_stStandardModuleItf.q_sDiagExt		:= FC_EtDiagExtToString(i_etDiagExt := ET_DiagExt.WaitCmdsDone);
			TPL.ET_DiagExt.WaitForCmd : 
				iq_stStandardModuleItf.q_udiDiagExt	:= ET_DiagExt.WaitForCmd;
				iq_stStandardModuleItf.q_sDiagExt		:= FC_EtDiagExtToString(i_etDiagExt := ET_DiagExt.WaitForCmd);
			ELSE
				iq_stStandardModuleItf.q_etDiag		:= GD. ET_Diag.UnexpectedProgramBehavior;
				iq_stStandardModuleItf.q_udiDiagExt	:= ET_DiagExt.UnknownStateModuleController;
				iq_stStandardModuleItf.q_sDiagExt		:= FC_EtDiagExtToString(i_etDiagExt := ET_DiagExt.UnknownStateModuleController);
		END_CASE
	ELSE
		iq_stStandardModuleItf.q_etDiag		:= GD.ET_Diag.DiagActive;
		iq_stStandardModuleItf.q_udiDiagExt	:= ET_DiagExt.ModuleControllerException;
		iq_stStandardModuleItf.q_sDiagExt		:= FC_EtDiagExtToString(i_etDiagExt := ET_DiagExt.ModuleControllerException);
		iq_stStandardModuleItf.q_sMsg			:= PDL.FC_MultiConcat(	i_sString1 := GD.FC_EtDiagToString(i_etDiag := etDiagModuleController), 
																			i_sString2 := ' - ',
																			i_sString3 := TPL.FC_EtDiagExtToString(i_etDiagExt := etDiagExtModuleController), 
																			i_sString4 := '');
	END_IF
END_IF

(* End of system generated code, only to be changed by experienced programmers *)
END_ACTION

ACTION Start_Action:
(* This step is active until the machine is being enabled *)

(* System generated code, do not change without consulting 'Schneider Electric Automation GmbH' - otherwise you risk instability!!! *)
iq_stStandardModuleItf.q_xActive			:= FALSE;
iq_stStandardModuleItf.q_xReady			:= FALSE;

iq_stStandardModuleItf.q_etDiag			:= GD.ET_Diag.Ok;
iq_stStandardModuleItf.q_udiDiagExt		:= ET_DiagExt.Disabled;
iq_stStandardModuleItf.q_sDiagExt			:= FC_EtDiagExtToString(i_etDiagExt := iq_stStandardModuleItf.q_udiDiagExt);
iq_stStandardModuleItf.q_sMsg				:= '';

iq_stStandardModuleItf.q_dwModuleType		:= TPL.ET_ModuleType.NodeModule;
iq_stStandardModuleItf.q_sModuleTypeName	:= 'NodeModule';
iq_stStandardModuleItf.q_udiModuleVersion	:= 1;	
(* End of system generated code, do not change without consulting 'Schneider Electric Automation GmbH' - otherwise you risk instability!!! *)

(* System generated code, to be changed by experienced programmers *)
IF iq_stStandardModuleItf.iq_diCMD <> 0 AND NOT iq_stStandardModuleItf.i_xEnable THEN
	iq_stStandardModuleItf.iq_diCMD := 0;
END_IF
(* End of system generated code, to be changed by experienced programmers *)

(* Application specific code *)
(* ToDo: Add your application specific code here *)
;
(* End of application specific code *)
END_ACTION

ACTION SubModules_Action:
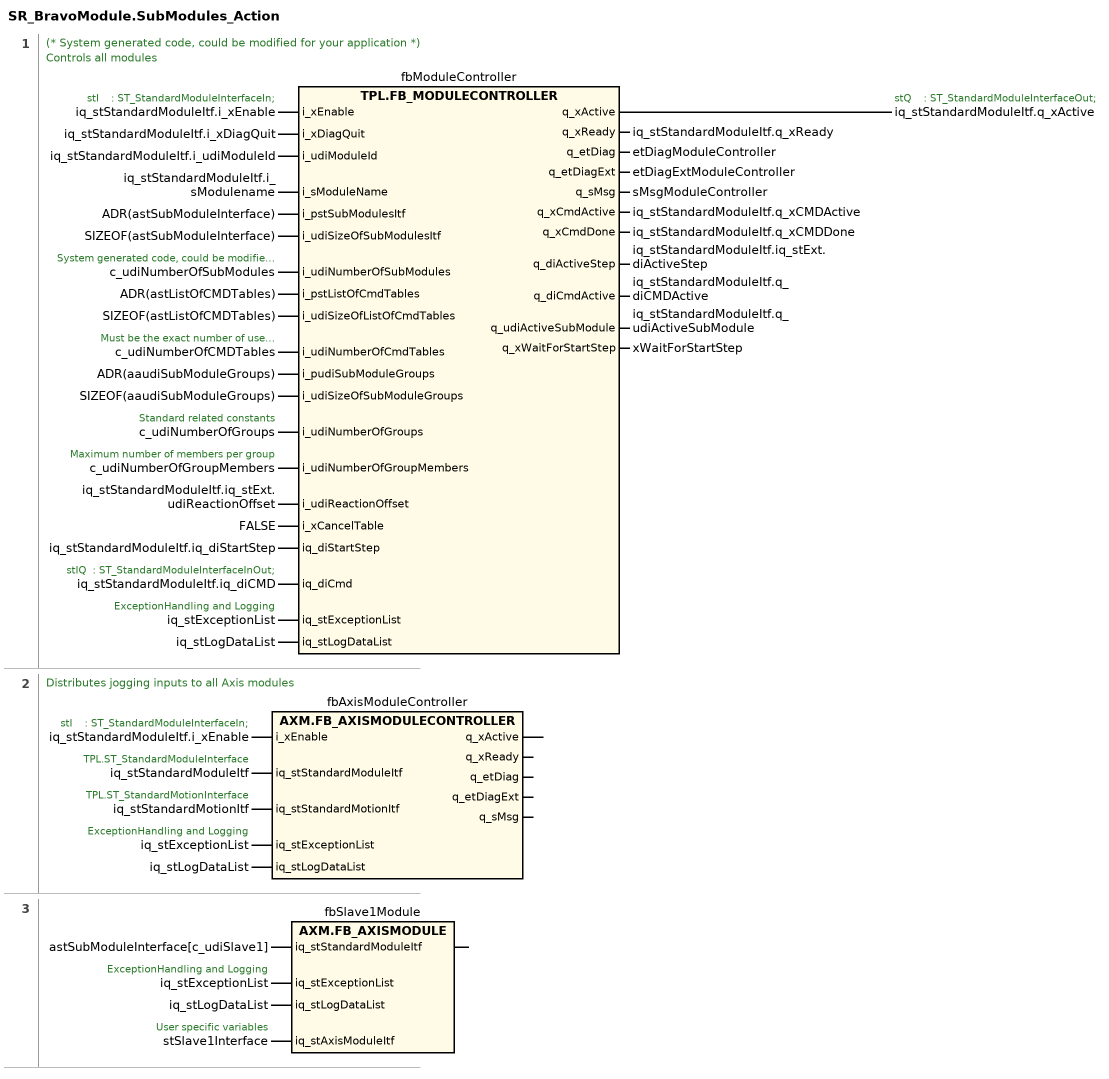
// NETWORK 1
// 					(* System generated code, could be modified for your application *)
// Controls all modules
//
//   fbModuleController: Modules related variables
//   iq_stStandardModuleItf.i_xEnable: stI : ST_StandardModuleInterfaceIn;
//   c_udiNumberOfSubModules: System generated code, could be modified for your application
//   c_udiNumberOfCMDTables: Must be the exact number of used CMDTables!
//   c_udiNumberOfGroups: Standard related constants
//   c_udiNumberOfGroupMembers: Maximum number of members per group
//   iq_stStandardModuleItf.iq_diCMD: stIQ : ST_StandardModuleInterfaceInOut;
//   iq_stExceptionList: ExceptionHandling and Logging
//   iq_stStandardModuleItf.q_xActive: stQ : ST_StandardModuleInterfaceOut;
fbModuleController(
    i_xEnable := iq_stStandardModuleItf.i_xEnable,
    i_xDiagQuit := iq_stStandardModuleItf.i_xDiagQuit,
    i_udiModuleId := iq_stStandardModuleItf.i_udiModuleId,
    i_sModuleName := iq_stStandardModuleItf.i_sModulename,
    i_pstSubModulesItf := ADR(astSubModuleInterface),
    i_udiSizeOfSubModulesItf := SIZEOF(astSubModuleInterface),
    i_udiNumberOfSubModules := c_udiNumberOfSubModules,
    i_pstListOfCmdTables := ADR(astListOfCMDTables),
    i_udiSizeOfListOfCmdTables := SIZEOF(astListOfCMDTables),
    i_udiNumberOfCmdTables := c_udiNumberOfCMDTables,
    i_pudiSubModuleGroups := ADR(aaudiSubModuleGroups),
    i_udiSizeOfSubModuleGroups := SIZEOF(aaudiSubModuleGroups),
    i_udiNumberOfGroups := c_udiNumberOfGroups,
    i_udiNumberOfGroupMembers := c_udiNumberOfGroupMembers,
    i_udiReactionOffset := iq_stStandardModuleItf.iq_stExt.udiReactionOffset,
    i_xCancelTable := FALSE,
    iq_diStartStep := iq_stStandardModuleItf.iq_diStartStep,
    iq_diCmd := iq_stStandardModuleItf.iq_diCMD,
    iq_stExceptionList := iq_stExceptionList,
    iq_stLogDataList := iq_stLogDataList,
    q_xReady => iq_stStandardModuleItf.q_xReady,
    q_etDiag => etDiagModuleController,
    q_etDiagExt => etDiagExtModuleController,
    q_sMsg => sMsgModuleController,
    q_xCmdActive => iq_stStandardModuleItf.q_xCMDActive,
    q_xCmdDone => iq_stStandardModuleItf.q_xCMDDone,
    q_diActiveStep => iq_stStandardModuleItf.iq_stExt.diActiveStep,
    q_diCmdActive => iq_stStandardModuleItf.q_diCMDActive,
    q_udiActiveSubModule => iq_stStandardModuleItf.q_udiActiveSubModule,
    q_xWaitForStartStep => xWaitForStartStep); // TPL.FB_MODULECONTROLLER
iq_stStandardModuleItf.q_xActive := fbModuleController.q_xActive;

// NETWORK 2
// Distributes jogging inputs to all Axis modules
//   iq_stStandardModuleItf.i_xEnable: stI : ST_StandardModuleInterfaceIn;
//   iq_stStandardModuleItf: TPL.ST_StandardModuleInterface
//   iq_stStandardMotionItf: TPL.ST_StandardMotionInterface
//   iq_stExceptionList: ExceptionHandling and Logging
fbAxisModuleController(
    i_xEnable := iq_stStandardModuleItf.i_xEnable,
    iq_stStandardModuleItf := iq_stStandardModuleItf,
    iq_stStandardMotionItf := iq_stStandardMotionItf,
    iq_stExceptionList := iq_stExceptionList,
    iq_stLogDataList := iq_stLogDataList); // AXM.FB_AXISMODULECONTROLLER

// NETWORK 3
//   iq_stExceptionList: ExceptionHandling and Logging
//   stSlave1Interface: User specific variables
fbSlave1Module(
    iq_stStandardModuleItf := astSubModuleInterface[c_udiSlave1],
    iq_stExceptionList := iq_stExceptionList,
    iq_stLogDataList := iq_stLogDataList,
    iq_stAxisModuleItf := stSlave1Interface); // AXM.FB_AXISMODULE

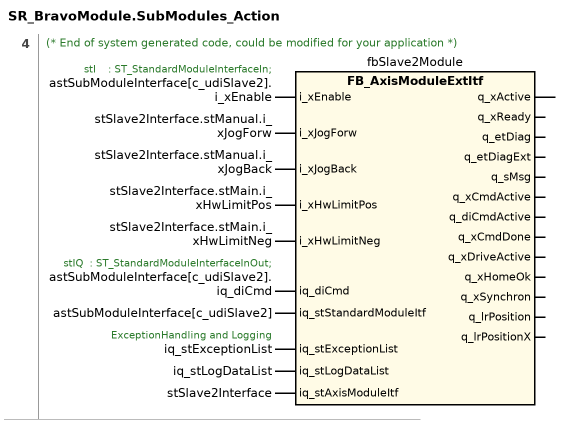
// NETWORK 4
// (* End of system generated code, could be modified for your application *)
//   astSubModuleInterface[c_udiSlave2].i_xEnable: stI : ST_StandardModuleInterfaceIn;
//   astSubModuleInterface[c_udiSlave2].iq_diCmd: stIQ : ST_StandardModuleInterfaceInOut;
//   iq_stExceptionList: ExceptionHandling and Logging
fbSlave2Module(
    i_xEnable := astSubModuleInterface[c_udiSlave2].i_xEnable,
    i_xJogForw := stSlave2Interface.stManual.i_xJogForw,
    i_xJogBack := stSlave2Interface.stManual.i_xJogBack,
    i_xHwLimitPos := stSlave2Interface.stMain.i_xHwLimitPos,
    i_xHwLimitNeg := stSlave2Interface.stMain.i_xHwLimitNeg,
    iq_diCmd := astSubModuleInterface[c_udiSlave2].iq_diCmd,
    iq_stStandardModuleItf := astSubModuleInterface[c_udiSlave2],
    iq_stExceptionList := iq_stExceptionList,
    iq_stLogDataList := iq_stLogDataList,
    iq_stAxisModuleItf := stSlave2Interface); // FB_AxisModuleExtItf
END_ACTION

ACTION UpdateStructs:
(* System generated code, do not change without consulting 'Schneider Electric Automation GmbH' - otherwise you risk instability!!!*)
fbDetectOnlineChange(	i_xEnable	:= TRUE, 
						i_xDetect	:= TRUE, 
						q_xActive	=> xDetectOnlineChangeActive, 
						q_xReady	=> xDetectOnlineChangeReady, 
						q_etDiag	=> etDetectOnlineChangeDiag, 
						q_etDiagExt	=> etDetectOnlineChangeDiagExt, 
						q_sMsg		=> sDetectOnlineChangeMsg, 
						q_xChange	=> );
						
IF(NOT fbDetectOnlineChange.q_xChange) THEN
	RETURN;
END_IF

iq_stStandardModuleItf.iq_stExt.udiNumberOfSubModules 		:= c_udiNumberOfSubModules;
iq_stStandardModuleItf.iq_stExt.dwSubModulesItf		 		:= ADR(astSubModuleInterface);
iq_stStandardModuleItf.iq_stExt.pdwSubModulesAddItf		 	:= ADR(adwSubModuleAddInterfaces);
iq_stStandardModuleItf.iq_stExt.pstListofCMDTables			:= ADR(astListOfCMDTables);
iq_stStandardModuleItf.iq_stExt.udiNumberOfCmdTables		:= c_udiNumberOfCMDTables;
(* End of system generated code, do not change without consulting 'Schneider Electric Automation GmbH' - otherwise you risk instability!!!*)

(* System generated code, could be modified for your application *)
xUpdateStructsException := FALSE;

(*****************************************************************************************************************************************************)
(* Update CmdTable - Prepare *)

TPL.FC_UpdateCmdTableListElement(	i_pstListofCMDTables	:= ADR(astListofCMDTables),
									i_udiNumberOfCmdTables	:= c_udiNumberOfCMDTables,
									i_diCMD					:= ET_Cmd.Prepare,
									i_pstCMDTable			:= ADR(astPrepareTable),
									q_etDiag				=> etDiag,
									q_etDiagExt				=> etDiagExtTPL);
									
IF etDiag <> GD.ET_Diag.Ok AND NOT xUpdateStructsException THEN
	xUpdateStructsException := TRUE;
	
	stUpdateStructsException.sMsg := PDL.FC_MultiConcat(i_sString1 := 'Update CmdTable: Prepare - ', 
														i_sString2 := GD.FC_EtDiagToString(i_etDiag := etDiag), 
														i_sString3 := ' - ', 
														i_sString4 := TPL.FC_EtDiagExtToString(i_etDiagExt := etDiagExtTPL));
END_IF										

(*****************************************************************************************************************************************************)
(* Update CmdTable - Auto *)

TPL.FC_UpdateCmdTableListElement(	i_pstListofCMDTables	:= ADR(astListofCMDTables),
									i_udiNumberOfCmdTables	:= c_udiNumberOfCMDTables,
									i_diCMD					:= ET_Cmd.Auto,
									i_pstCMDTable			:= ADR(astAutoTable),
									q_etDiag				=> etDiag,
									q_etDiagExt				=> etDiagExtTPL);
									
IF etDiag <> GD.ET_Diag.Ok AND NOT xUpdateStructsException THEN
	xUpdateStructsException := TRUE;
	
	stUpdateStructsException.sMsg := PDL.FC_MultiConcat(i_sString1 := 'Update CmdTable: Auto - ', 
														i_sString2 := GD.FC_EtDiagToString(i_etDiag := etDiag), 
														i_sString3 := ' - ', 
														i_sString4 := TPL.FC_EtDiagExtToString(i_etDiagExt := etDiagExtTPL));
END_IF		

(*****************************************************************************************************************************************************)
(* Update CmdTable - Manual *)

TPL.FC_UpdateCmdTableListElement(	i_pstListofCMDTables	:= ADR(astListofCMDTables),
									i_udiNumberOfCmdTables	:= c_udiNumberOfCMDTables,
									i_diCMD					:= ET_Cmd.Manual,
									i_pstCMDTable			:= ADR(astManualTable),
									q_etDiag				=> etDiag,
									q_etDiagExt				=> etDiagExtTPL);
									
IF etDiag <> GD.ET_Diag.Ok AND NOT xUpdateStructsException THEN
	xUpdateStructsException := TRUE;
	
	stUpdateStructsException.sMsg := PDL.FC_MultiConcat(i_sString1 := 'Update CmdTable: Manual - ', 
														i_sString2 := GD.FC_EtDiagToString(i_etDiag := etDiag), 
														i_sString3 := ' - ', 
														i_sString4 := TPL.FC_EtDiagExtToString(i_etDiagExt := etDiagExtTPL));
END_IF		

(*****************************************************************************************************************************************************)
(* Update CmdTable - Stop *)

TPL.FC_UpdateCmdTableListElement(	i_pstListofCMDTables	:= ADR(astListofCMDTables),
									i_udiNumberOfCmdTables	:= c_udiNumberOfCMDTables,
									i_diCMD					:= ET_Cmd.Stop,
									i_pstCMDTable			:= ADR(astStopTable),
									q_etDiag				=> etDiag,
									q_etDiagExt				=> etDiagExtTPL);
									
IF etDiag <> GD.ET_Diag.Ok AND NOT xUpdateStructsException THEN
	xUpdateStructsException := TRUE;
	
	stUpdateStructsException.sMsg := PDL.FC_MultiConcat(i_sString1 := 'Update CmdTable: Stop - ', 
														i_sString2 := GD.FC_EtDiagToString(i_etDiag := etDiag), 
														i_sString3 := ' - ', 
														i_sString4 := TPL.FC_EtDiagExtToString(i_etDiagExt := etDiagExtTPL));
END_IF		

(*****************************************************************************************************************************************************)
(* Update CmdTable - Start *)

TPL.FC_UpdateCmdTableListElement(	i_pstListofCMDTables	:= ADR(astListofCMDTables),
									i_udiNumberOfCmdTables	:= c_udiNumberOfCMDTables,
									i_diCMD					:= ET_Cmd.Start,
									i_pstCMDTable			:= ADR(astStartTable),
									q_etDiag				=> etDiag,
									q_etDiagExt				=> etDiagExtTPL);
									
IF etDiag <> GD.ET_Diag.Ok AND NOT xUpdateStructsException THEN
	xUpdateStructsException := TRUE;
	
	stUpdateStructsException.sMsg := PDL.FC_MultiConcat(i_sString1 := 'Update CmdTable: Start - ', 
														i_sString2 := GD.FC_EtDiagToString(i_etDiag := etDiag), 
														i_sString3 := ' - ', 
														i_sString4 := TPL.FC_EtDiagExtToString(i_etDiagExt := etDiagExtTPL));
END_IF		

(*****************************************************************************************************************************************************)
(* Update CmdTable - Abort *)

TPL.FC_UpdateCmdTableListElement(	i_pstListofCMDTables	:= ADR(astListofCMDTables),
									i_udiNumberOfCmdTables	:= c_udiNumberOfCMDTables,
									i_diCMD					:= ET_Cmd.Abort,
									i_pstCMDTable			:= ADR(astAbortTable),
									q_etDiag				=> etDiag,
									q_etDiagExt				=> etDiagExtTPL);
									
IF etDiag <> GD.ET_Diag.Ok AND NOT xUpdateStructsException THEN
	xUpdateStructsException := TRUE;
	
	stUpdateStructsException.sMsg := PDL.FC_MultiConcat(i_sString1 := 'Update CmdTable: Abort - ', 
														i_sString2 := GD.FC_EtDiagToString(i_etDiag := etDiag), 
														i_sString3 := ' - ', 
														i_sString4 := TPL.FC_EtDiagExtToString(i_etDiagExt := etDiagExtTPL));
END_IF		

(*****************************************************************************************************************************************************)
(* Update CmdTable - Hold *)

TPL.FC_UpdateCmdTableListElement(	i_pstListofCMDTables	:= ADR(astListofCMDTables),
									i_udiNumberOfCmdTables	:= c_udiNumberOfCMDTables,
									i_diCMD					:= ET_Cmd.Hold,
									i_pstCMDTable			:= ADR(astHoldTable),
									q_etDiag				=> etDiag,
									q_etDiagExt				=> etDiagExtTPL);
									
IF etDiag <> GD.ET_Diag.Ok AND NOT xUpdateStructsException THEN
	xUpdateStructsException := TRUE;
	
	stUpdateStructsException.sMsg := PDL.FC_MultiConcat(i_sString1 := 'Update CmdTable: Hold - ', 
														i_sString2 := GD.FC_EtDiagToString(i_etDiag := etDiag), 
														i_sString3 := ' - ', 
														i_sString4 := TPL.FC_EtDiagExtToString(i_etDiagExt := etDiagExtTPL));
END_IF		

(*****************************************************************************************************************************************************)
(* Update CmdTable - BrakeRelease *)

TPL.FC_UpdateCmdTableListElement(	i_pstListofCMDTables	:= ADR(astListofCMDTables),
									i_udiNumberOfCmdTables	:= c_udiNumberOfCMDTables,
									i_diCMD					:= ET_Cmd.BrakeRelease,
									i_pstCMDTable			:= ADR(astBrakeReleaseTable),
									q_etDiag				=> etDiag,
									q_etDiagExt				=> etDiagExtTPL);
									
IF etDiag <> GD.ET_Diag.Ok AND NOT xUpdateStructsException THEN
	xUpdateStructsException := TRUE;
	
	stUpdateStructsException.sMsg := PDL.FC_MultiConcat(i_sString1 := 'Update CmdTable: BrakeRelease - ', 
														i_sString2 := GD.FC_EtDiagToString(i_etDiag := etDiag), 
														i_sString3 := ' - ', 
														i_sString4 := TPL.FC_EtDiagExtToString(i_etDiagExt := etDiagExtTPL));
END_IF		
									
(*****************************************************************************************************************************************************)
(* Update AddInterface - Slave1 *)

AXM.FC_UpdateAddInterfaceStruct(	i_pdwSubModuleAddInterfaces	:= ADR(adwSubModuleAddInterfaces),
									i_udiSubModuleConstant		:= c_udiSlave1,
									iq_stAxisModuleItf			:= stSlave1Interface,
									q_etDiag					=> etDiag,
									q_etDiagExt					=> etDiagExtAXM);
									
IF etDiag <> GD.ET_Diag.Ok AND NOT xUpdateStructsException THEN
	xUpdateStructsException := TRUE;
	
	stUpdateStructsException.sMsg := PDL.FC_MultiConcat(i_sString1 := 'Update AddInterface: Slave1 - ', 
														i_sString2 := GD.FC_EtDiagToString(i_etDiag := etDiag), 
														i_sString3 := ' - ', 
														i_sString4 := AXM.FC_EtDiagExtToString(i_etDiagExt := etDiagExtAXM));
END_IF		

(*****************************************************************************************************************************************************)
(* Update AddInterface - Slave2 *)

AXM.FC_UpdateAddInterfaceStruct(	i_pdwSubModuleAddInterfaces	:= ADR(adwSubModuleAddInterfaces),
									i_udiSubModuleConstant		:= c_udiSlave2,
									iq_stAxisModuleItf			:= stSlave2Interface,
									q_etDiag					=> etDiag,
									q_etDiagExt					=> etDiagExtAXM);
									
IF etDiag <> GD.ET_Diag.Ok AND NOT xUpdateStructsException THEN
	xUpdateStructsException := TRUE;
	
	stUpdateStructsException.sMsg := PDL.FC_MultiConcat(i_sString1 := 'Update AddInterface: Slave2 - ', 
														i_sString2 := GD.FC_EtDiagToString(i_etDiag := etDiag), 
														i_sString3 := ' - ', 
														i_sString4 := AXM.FC_EtDiagExtToString(i_etDiagExt := etDiagExtAXM));
END_IF		

(*****************************************************************************************************************************************************)
(* Set exception if any exception occurred *)

TPL.FC_SetException(i_xExceptionActive	:= xUpdateStructsException, 
					iq_stException		:= stUpdateStructsException, 
					iq_stExceptionList	:= iq_stExceptionList, 
					iq_stLogDataList	:= iq_stLogDataList);
					
xInitSuccessful := xInitSuccessful AND NOT xUpdateStructsException;

etDiag := GD.ET_Diag.Ok;
(* End of system generated code, could be modified for your application *)
END_ACTION

END_PROGRAM

// LMC_PacDrive/Application/CrankModuleExample/Examples/ExampleModulesExtItf/FB_AxisModuleExtItf
FUNCTION_BLOCK FB_AxisModuleExtItf

VAR_INPUT
(* Part of TPL.ST_StandardModuleInterface.i_... *)
	i_xEnable		: BOOL;
	
(* Part of AXM.ST_ModuleInterface.stManual.i_... *)
	i_xJogForw		: BOOL;
	i_xJogBack		: BOOL;
	
(* Part of AXM.ST_ModuleInterface.stMain.i_... *)
	i_xHwLimitPos	: BOOL;
	i_xHwLimitNeg	: BOOL;
END_VAR

VAR_IN_OUT
(* Part of TPL.ST_StandardModuleInterface.iq_... *)	
	iq_diCmd				: DINT;

(* TPL.ST_StandardModuleInterface *)		
	iq_stStandardModuleItf	: TPL.ST_StandardModuleInterface;
	
(* ExceptionHandling and Logging *)	
	iq_stExceptionList		: TPL.ST_ExceptionList;
	iq_stLogDataList		: TPL.ST_LogDataList;
	
(* AXM.ST_ModuleInterface *)
	iq_stAxisModuleItf		: AXM.ST_ModuleInterface;
END_VAR

VAR_OUTPUT
(* Part of TPL.ST_StandardModuleInterface.q_... *)	
	q_xActive		: BOOL;
	q_xReady		: BOOL;
	q_etDiag		: GD.ET_Diag := GD.ET_Diag.Ok;
	q_etDiagExt		: AXM.ET_DiagExt := AXM.ET_DiagExt.Disabled;
	q_sMsg			: STRING[80] := '';
	q_xCmdActive	: BOOL;
	q_diCmdActive	: DINT;
	q_xCmdDone		: BOOL;
	
(* Part of AXM.ST_ModuleInterface.stMain.q_... *)
	q_xDriveActive	: BOOL;
	q_xHomeOk		: BOOL;
	q_xSynchron		: BOOL;
	q_lrPosition	: LREAL;
	q_lrPositionX	: LREAL;
END_VAR

VAR
	fbAxisModule : AXM.FB_AxisModule;
END_VAR

(* System generated code, could be modified for your application *)

iq_stStandardModuleItf.i_xEnable	:= i_xEnable;
iq_stStandardModuleItf.iq_diCmd		:= iq_diCmd;

iq_stAxisModuleItf.stMain.i_xHwLimitPos	:= i_xHwLimitPos;
iq_stAxisModuleItf.stMain.i_xHwLimitNeg	:= i_xHwLimitNeg;

iq_stAxisModuleItf.stManual.i_xJogForw	:= i_xJogForw;
iq_stAxisModuleItf.stManual.i_xJogBack	:= i_xJogBack;

(* Module call *)
fbAxisModule(	iq_stStandardModuleItf	:= iq_stStandardModuleItf,
				iq_stExceptionList		:= iq_stExceptionList,
				iq_stLogDataList		:= iq_stLogDataList,
				iq_stAxisModuleItf		:= iq_stAxisModuleItf);
				
iq_diCmd := iq_stStandardModuleItf.iq_diCmd;

q_xActive		:= iq_stStandardModuleItf.q_xActive;
q_xReady		:= iq_stStandardModuleItf.q_xReady;
q_etDiag		:= iq_stStandardModuleItf.q_etDiag;
q_etDiagExt		:= iq_stStandardModuleItf.q_udiDiagExt;
q_sMsg			:= iq_stStandardModuleItf.q_sMsg;
q_xCmdActive	:= iq_stStandardModuleItf.q_xCmdActive;
q_diCmdActive	:= iq_stStandardModuleItf.q_diCmdActive;
q_xCmdDone		:= iq_stStandardModuleItf.q_xCmdDone;

q_xDriveActive	:= iq_stAxisModuleItf.stMain.q_xDriveActive;
q_xHomeOk		:= iq_stAxisModuleItf.stMain.q_xHomeOk;
q_xSynchron		:= iq_stAxisModuleItf.stMain.q_xSynchron;
q_lrPosition	:= iq_stAxisModuleItf.stMain.q_lrPosition;
q_lrPositionX	:= iq_stAxisModuleItf.stMain.q_lrPositionX;

(* End of system generated code, could be modified for your application *)

END_FUNCTION_BLOCK

// LMC_PacDrive/Application/CrankModuleExample/Examples/ExampleModulesExtItf/SR_CharlyModuleExtItf
PROGRAM SR_CharlyModuleExtItf

VAR_INPUT
(* Part of TPL.ST_StandardModuleInterface.i_... *)
	i_xEnable						: BOOL;
	
(* Master of AlphaModule *)
	i_ifMaster						: SystemConfigurationItf.IF_Master;
END_VAR

VAR_IN_OUT
(* Part of TPL.ST_StandardModuleInterface.iq_... *)
	iq_diCmd						: DINT;
	iq_diStartStep					: DINT;

(* TPL.ST_StandardModuleInterface *)	
	iq_stStandardModuleItf			: TPL.ST_StandardModuleInterface;
	
(* TPL.ST_StandardMotionInterface *)		
	iq_stStandardMotionItf			: TPL.ST_StandardMotionInterface;
	
(* ExceptionHandling and Logging *)	
	iq_stExceptionList				: TPL.ST_ExceptionList;
	iq_stLogDataList				: TPL.ST_LogDataList;
END_VAR

VAR_OUTPUT
(* Part of TPL.ST_StandardModuleInterface.q_... *)
	q_xActive						: BOOL;
	q_xReady						: BOOL;
	q_etDiag						: GD.ET_Diag; 
	q_etDiagExt						: ET_DiagExt;
	q_sMsg							: STRING[80];	
	q_xCmdActive					: BOOL;
	q_diCmdActive					: DINT;
	q_xCmdDone						: BOOL;
	q_udiActiveSubModule			: UDINT;
	q_udiSubModuleInException		: UDINT;
END_VAR

(* System generated code, could be modified for your application *)

iq_stStandardModuleItf.i_xEnable		:= i_xEnable;
iq_stStandardModuleItf.iq_diCmd			:= iq_diCmd;
iq_stStandardModuleItf.iq_diStartStep	:= iq_diStartStep;

(* Module call *)
SR_CharlyModule(i_ifMaster				:= i_ifMaster, 
				iq_stStandardModuleItf	:= iq_stStandardModuleItf, 
				iq_stStandardMotionItf	:= iq_stStandardMotionItf, 
				iq_stExceptionList		:= iq_stExceptionList, 
				iq_stLogDataList		:= iq_stLogDataList);
				
iq_diCmd		:= iq_stStandardModuleItf.iq_diCmd;
iq_diStartStep	:= iq_stStandardModuleItf.iq_diStartStep;

q_xActive						:= iq_stStandardModuleItf.q_xActive;
q_xReady						:= iq_stStandardModuleItf.q_xReady;
q_etDiag						:= iq_stStandardModuleItf.q_etDiag; 
q_etDiagExt						:= iq_stStandardModuleItf.q_udiDiagExt;
q_sMsg							:= iq_stStandardModuleItf.q_sMsg;	
q_xCmdActive					:= iq_stStandardModuleItf.q_xCmdActive;
q_diCmdActive					:= iq_stStandardModuleItf.q_diCmdActive;
q_xCmdDone						:= iq_stStandardModuleItf.q_xCmdDone;
q_udiActiveSubModule			:= iq_stStandardModuleItf.q_udiActiveSubModule;
q_udiSubModuleInException		:= iq_stStandardModuleItf.q_udiSubModuleInException;

(* End of system generated code, could be modified for your application *)

END_PROGRAM

// LMC_PacDrive/Application/CrankModuleExample/EquipmentModules/SR_CharlyModule
PROGRAM SR_CharlyModule

VAR CONSTANT
(* Standard related constants *)
	c_udiNumberOfGroups				: UDINT := 3;			(* Maximum number of groups *)
	c_udiNumberOfGroupMembers		: UDINT := 10;			(* Maximum number of members per group *)

	c_udiNumberOfCmdTables			: UDINT := 8;			(* Must be the exact number of used CMDTables!*)
	c_udiNumberOfCmdSteps			: UDINT := 16;			(* Make sure that the number of commands/ Steps  that each table
																   contains does not exceed the c_diNumberOfCMDSteps variable.*)

(* Definition group of modules *)
	c_udiCharlyGroup1				: UDINT := 2001;		(* Name of module group  1 *)
	c_udiCharlyGroup2				: UDINT := 2002;		(* Name of module group  2 *)

